// TwinCAT 3 PLC project Katzenhofer
// ProgramVersion: 3.1.4023.0
// libraries:
//   EfficientIO Energy Basic, * (EfficientIO)
//   EfficientIO ModbusTCP, * (EfficientIO)
//   Lynus Persistent Data V1, * (Lynus AG)
//   Lynus Standards, * (EfficientIO)
//   Tc2_IoFunctions, * (Beckhoff Automation GmbH)
//   Tc2_ModbusSrv, * (Beckhoff Automation GmbH)
//   Tc2_Standard, * (Beckhoff Automation GmbH)
//   Tc2_System, * (Beckhoff Automation GmbH)
//   Tc2_Utilities, * (Beckhoff Automation GmbH)
//   Tc3_Module, * (Beckhoff Automation GmbH)
//   EfficientIO Communicator,newest,EfficientIO
// project tree:
//   / FastTask.TcTTO (not stored), MiddleTask.TcTTO, SlowTask.TcTTO
//   FB/ FB_IntervalBit.TcPOU (not stored), FB_ModBus_100Registers_FC3.TcPOU, FB_ModBus_100Registers_FC3_inclID.TcPOU
//   POUs/ prgBattery.TcPOU, prgCalc.TcPOU, prgComEffIO.TcPOU, prgCS.TcPOU, prgEM.TcPOU, prgEMS.TcPOU, prgGrid.TcPOU, prgPersistent.TcPOU, prgPV.TcPOU, prgRWEffIO.TcPOU, prgVarEffIO.TcPOU
// real-time tasks:
//   TASK FastTask: cycle T#5ms, priority 6, ADS port 350
//   TASK MiddleTask: cycle T#10ms, priority 8, ADS port 351
//   TASK SlowTask: cycle T#20ms, priority 10, ADS port 352
// I/O:
//   DEVICE Device 1 (Beckhoff CCAT)
//   DEVICE Device 2 (CX-BK)
//     Box 1 (CX-BK)
// variable links:
//   Katzenhofer/Katzenhofer Instance <-> Device 2 (CX-BK)/Box 1 (CX-BK)
//     MiddleTask Inputs/prgEM.fbEM1.fbKL3403.byStateCH1 <-> Term 2 (KL3403)/Channel 1/State
//     MiddleTask Inputs/prgEM.fbEM1.fbKL3403.byStateCH2 <-> Term 2 (KL3403)/Channel 2/State
//     MiddleTask Inputs/prgEM.fbEM1.fbKL3403.byStateCH3 <-> Term 2 (KL3403)/Channel 3/State
//     MiddleTask Inputs/prgEM.fbEM1.fbKL3403.iDataInCH1 <-> Term 2 (KL3403)/Channel 1/Data In
//     MiddleTask Inputs/prgEM.fbEM1.fbKL3403.iDataInCH2 <-> Term 2 (KL3403)/Channel 2/Data In
//     MiddleTask Inputs/prgEM.fbEM1.fbKL3403.iDataInCH3 <-> Term 2 (KL3403)/Channel 3/Data In
//     MiddleTask Inputs/prgEM.fbKBusState.uiKBusState_OUT <-> Inputs/State
//     MiddleTask Outputs/prgEM.fbEM1.fbKL3403.byCntrCH1 <-> Term 2 (KL3403)/Channel 1/Ctrl
//     MiddleTask Outputs/prgEM.fbEM1.fbKL3403.byCntrCH2 <-> Term 2 (KL3403)/Channel 2/Ctrl
//     MiddleTask Outputs/prgEM.fbEM1.fbKL3403.byCntrCH3 <-> Term 2 (KL3403)/Channel 3/Ctrl

CONFIGURATION Katzenhofer
    RESOURCE PLC ON TwinCAT3
        TASK MiddleTask(INTERVAL := T#10ms, PRIORITY := 8);
        TASK SlowTask(INTERVAL := T#20ms, PRIORITY := 10);
        PROGRAM prgEMS WITH MiddleTask : prgEMS;
        PROGRAM prgPersistent WITH MiddleTask : prgPersistent;
        PROGRAM prgPV WITH MiddleTask : prgPV;
        PROGRAM prgBattery WITH MiddleTask : prgBattery;
        PROGRAM prgEM WITH MiddleTask : prgEM;
        PROGRAM prgGrid WITH MiddleTask : prgGrid;
        PROGRAM prgCS WITH MiddleTask : prgCS;
        PROGRAM prgCalc WITH MiddleTask : prgCalc;
        PROGRAM prgComEffIO WITH SlowTask : prgComEffIO;
    END_RESOURCE
END_CONFIGURATION

// ---- POUs/prgEMS.TcPOU
PROGRAM prgEMS
VAR PERSISTENT
	byMaxDepthOfDischrgEPO		: BYTE;							//{#lynus.ag#()}
	byPrioMinChrgBattSOCInEPO	: BYTE;							//{#lynus.ag#()}
	byResChrgfromGridToBatt		: BYTE;							//{#lynus.ag#()}
	byReserveSOCEPO				: BYTE;							//{#lynus.ag#()}
	uiUpdateTime				: UINT;							//{#lynus.ag#()}
	bEnableEMS					: BOOL;							//{#lynus.ag#()}
	bAllowChrgFromGrid			: BOOL;							//{#lynus.ag#()}
	rMainFuseCSEMS				: REAL;							//{#lynus.ag#()}
	iOperationModeEMS			: INT;							//{#lynus.ag#()}
	by_MinSOC_AdaptiveLC		: BYTE;							//{#lynus.ag#()}
END_VAR
VAR
	fbEMS						: FB_EMS_V12;
	bIsEnableEMS				: BOOL;							//{#lynus.ag#()}
	bStateAllowChrgFromGrid		: BOOL;							//{#lynus.ag#()}
	bHPActivate					: BOOL;							//{#lynus.ag#()}
	bControllingState			: BOOL;							//{#lynus.ag#()}
	iMessageEMS					: INT;							//{#lynus.ag#()}
	rHeartbeatEMS				: REAL;							//{#lynus.ag#()}
	rErrorWarningEMS			: REAL;							//{#lynus.ag#()}
	rReadyEMS					: REAL;							//{#lynus.ag#()}
	rNewBatteryPowerEMS			: REAL;							//{#lynus.ag#()}
	fbRestart					: NT_Reboot;
	byte_test: BYTE;
	real_test: REAL;
	m_test: BOOL;
	lreal_Test: LREAL;
	m_test2: BOOL;
	by_test: BYTE;
	m_Test3: BOOL;
	m_ZeroPowerRegulationActive: BOOL:=FALSE;					//{#lynus.ag#()}
	m_Enable_Dynamic_LM: BOOL;
	timer_CarConnected_CSPowerlow: Ton;
	m_ByteTemp: BOOL;					//{#lynus.ag#()}
	dw_Test: DWORD;
	iOperationModeEMS_actual	: INT;							//{#lynus.ag#()}
END_VAR

fbEMS.stSetupEMS.bAllowChrgFromGrid := bAllowChrgFromGrid;
fbEMS.stSetupEMS.byMaxDepthOfDischrgEPO := byMaxDepthOfDischrgEPO;
fbEMS.stSetupEMS.byPrioMinChrgBattSOCInEPO := byPrioMinChrgBattSOCInEPO;
fbEMS.stSetupEMS.byResChrgfromGridToBatt := byResChrgfromGridToBatt;
fbEMS.stSetupEMS.byReserveSOCEPO := byReserveSOCEPO;
fbEMS.stSetupEMS.rSizeMainFuseCS := rMainFuseCSEMS;
fbEMS.stSetupEMS.uiUpdateTime := uiUpdateTime;


(*
IF m_Enable_Dynamic_LM THEN
	IF prgBattery.dwSOCBattery > byMinSOCdynamicLM AND NOT prgCS.bCarConnected THEN
		iOperationModeEMS := 1;		// Eigenbedarfsoptimierung
	ELSE
		iOperationModeEMS := 3;		// Lastmanagement
	END_IF  
END_IF
*)

IF iOperationModeEMS = 0 THEN fbEMS.eOperationMode_Ext := E_OperatingMode_EMS.eAllOff;
ELSIF iOperationModeEMS = 1 THEN fbEMS.eOperationMode_Ext := E_OperatingMode_EMS.eSelfConsumption;	
ELSIF iOperationModeEMS = 2 THEN fbEMS.eOperationMode_Ext := E_OperatingMode_EMS.ePeakLoadCapping;
ELSIF iOperationModeEMS = 3 THEN fbEMS.eOperationMode_Ext := E_OperatingMode_EMS.eLoadManagement;			
ELSIF iOperationModeEMS = 4 THEN fbEMS.eOperationMode_Ext := E_OperatingMode_EMS.eAdaptiveLoadControl;			

END_IF

fbEMS(
	bEnable:= bEnableEMS, 
	diNrOfEM_IN_ECS:= , 
	stSetupEMS:= , 
	eOperationMode_Ext:= , 
	eSpeedModeBackendController:= E_SpeedModeBackendController_EMS.eSlow, 
	eSpeedModeLocalController:= E_SpeedModeLocalController_EMS.eSlow,
	bZeroPowerRegulation := m_ZeroPowerRegulationActive,
	by_MinSOC_AdaptiveLC:= by_MinSOC_AdaptiveLC , 
	bActivateHP:= bHPActivate, 
	bControllingState:= TRUE, //bControllingState, 
	rHeartbeat:= rHeartbeatEMS, 
	rErrorWarning:= rErrorWarningEMS, 
	rEnergyOptReady:= rReadyEMS, 
	rNewBattPower:= rNewBatteryPowerEMS, 
	b_AnyCarConnected:= prgCS.bCarConnected, 
	eMessageEMS=> iMessageEMS, 
	bStateEnable=> bIsEnableEMS, 
	bStateAllowChrgFromGrid=> bStateAllowChrgFromGrid, 
	bMissingPowerData=> , 
	bSurplusAvailable=> , 
	byProgress=> , 
	uiState_OUT=> , 
	diNrOfEMS_OUT=> , 
	arrMinPrioReached=> , 
	arrMaxPrioReached=> );

	
iOperationModeEMS_actual := fbEMS.eOperationMode;
	
fbRestart(
	NETID:= , 
	DELAY:= , 
	START:= , 
	TMOUT:= , 
	BUSY=> , 
	ERR=> , 
	ERRID=> );
	

timer_CarConnected_CSPowerlow( 	IN := prgCS.bCarConnected AND prgCS.lrPowerCS < 2,	// required to get out of zero power regulation if a car is connected all night long
								PT := T#10M);
							
m_ZeroPowerRegulationActive := prgCS.bCarConnected AND NOT timer_CarConnected_CSPowerlow.Q;
	
// TEMP

real_test:= Lynus_Standards.GVL_Energy.stDataElectricChargingStations[1,1].rTargetPowerEMS;


//byte_test:=Lynus_Standards.GVL_Energy.stDataElectricChargingStations[1,1].byPriority;
 
//m_test:=Lynus_Standards.GVL_Energy.stDataElectricChargingStations[1,1].bEnabled; 
//Lynus_Standards.GVL_Energy.stDataElectricChargingStations[1,1].rTargetPowerEMS 
//Lynus_Standards.GVL_Energy.stDataElectricChargingStations[1,1].rTargetPowerEMS + rValuePercentToControllableDevices;
		
 lreal_Test:=fbEMS.lrPowerDiffFuseECS;
 
m_test2:=Lynus_Standards.GVL_Energy.stDataElectricChargingStations[1,1].bIsControllable;
by_test:=Lynus_Standards.GVL_Energy.stDataElectricChargingStations[1,1].byPriority;
//by_test:=Lynus_Standards.GVL_Energy.stDataElectricChargingStations[1,fbEMS.arrLPPrioZeroSetToZeroP[5]].byPriority;
by_test:= Lynus_Standards.GVL_Energy.stDataElectricChargingStations[1,1].byPriority; 
 
m_Test3:=Lynus_Standards.GVL_Energy.stDataElectricMeters[1].bEnabled ;

END_PROGRAM

// ---- POUs/prgCS.TcPOU
PROGRAM prgCS
VAR PERSISTENT
	bEnabledCS				: BOOL;									//{#lynus.ag#()}
	byPrioCS				: BYTE;									//{#lynus.ag#()}
	bySOC_E_CS				: BYTE;									//{#lynus.ag#()}
	bySOC_D_CS				: BYTE;									//{#lynus.ag#()}
	byMinPowerCS			: BYTE;									//{#lynus.ag#()}
	rMaxPowerCS				: REAL;									//{#lynus.ag#()}
	lrCounterCS				: LREAL;								//{#lynus.ag#()}
	byManualyTargetPower	: BYTE;									//{#lynus.ag#()}
	bManualyOn				: BOOL;									//{#lynus.ag#()}
END_VAR
VAR
	fbCS					: FB_ECS_Alpitronic_Hypercharger;
	fbCSCounter				: FB_EnergyCounter;
	bIsEnabledCS			: BOOL;									//{#lynus.ag#()}
	byErrorWarningCS		: BYTE;									//{#lynus.ag#()}
	byStateMinPowerCS		: BYTE;									//{#lynus.ag#()}
	rTargetPowerCS			: REAL;									//{#lynus.ag#()}
	bCarConnected			: BOOL;									//{#lynus.ag#()}
	rChrgTime				: REAL;									//{#lynus.ag#()}
	lrPowerCS				: LREAL;								//{#lynus.ag#()}
	bSManualyOn				: BOOL;									//{#lynus.ag#()}
	bySManualyTargetPower	: BYTE;									//{#lynus.ag#()}
	b_CS_ModbusFault		: BOOL;									//{#lynus.ag#()}
END_VAR

fbCS.stSetupECS.byDisableSOC := bySOC_D_CS;
fbCS.stSetupECS.byEnableSOC := bySOC_E_CS;
fbCS.stSetupECS.byPriority := byPrioCS;
fbCS.stSetupECS.rMaxPower := rMaxPowerCS;
fbCS.stSetupECS.byCSMinPower := byMinPowerCS;
fbCS.stSetupECS.bManualyOn := bManualyOn;
fbCS.stSetupECS.byManualyTargetPower := byManualyTargetPower;

fbCS(
	bEnable:= bEnabledCS, 
	bPowerDataInvers:= , 
	byUnitID:= 1,				//Allways 1 
	diNrOfEMS_IN:= prgEMS.fbEMS.diNrOfEMS_OUT, 
	diNrOfEM_IN_CS:= , 
	sIPAdress:= '10.11.90.140',			//192.168.0.100', 
	stSetupECS:= , 
	stDataECS=> , 
	diNrOfECS_OUT=> );

bIsEnabledCS := fbCS.stDataECS.bEnabled;
byStateMinPowerCS := fbCS.stDataECS.bySCSMinPower;
rTargetPowerCS := fbCS.stDataECS.rTargetPower;	
byErrorWarningCS := fbCS.stDataECS.byErrorWarning;
bCarConnected := fbCS.stDataECS.bCarConnected;
rChrgTime := fbCS.stDataECS.arrChargingTimeInMin[1];
lrPowerCS := fbCS.stDataECS.lrTotalPower;
bSManualyOn := fbCS.stDataECS.bSManualyOn;
bySManualyTargetPower := fbCS.stDataECS.bySManualyTargetPower;
						
// EnergyCounter
fbCSCounter(
	byActiveTariff:= 1, 
	lrPowerInput:= lrPowerCS, 
	lrTotalCounterEnergy_Consumption=> );
	
IF fbCSCounter.lrTotalCounterEnergy_Consumption > lrCounterCS THEN  	
	lrCounterCS := fbCSCounter.lrTotalCounterEnergy_Consumption;
END_IF

b_CS_ModbusFault := fbCS.bMBTCPError;

END_PROGRAM

// ---- POUs/prgPersistent.TcPOU
PROGRAM prgPersistent
VAR
	fbUSV		: FB_WritePersistentData_CX81xx;

	fb_Reboot		: NT_reboot;
	m_Reboot		: BOOL:=FALSE;

END_VAR

fbUSV(
	eSaveModeData:= eUSVSaveMode.eSaveWhenPowerfail, 
	bLoadPersistentDataOk=> , 
	bPowerFailDetect=> , 
	bError=> , 
	bySaveProcess=> , 
	dwStorageLast24h=> , 
	udiErrorCode=> );
	
	
		
fb_Reboot(	netid := '',
			delay := 2,
			start := m_Reboot);

END_PROGRAM

// ---- POUs/prgPV.TcPOU
PROGRAM prgPV
VAR
	fbPV					: FB_Symo_PV_Inverter_FLOAT_1_DM_30_Inverter;
	fbPV_2					: FB_Symo_PV_Inverter_FLOAT_1_DM_30_Inverter;
	fbPV_3					: FB_Symo_PV_Inverter_FLOAT_1_DM_30_Inverter;
	fbPV_4					: FB_Symo_PV_Inverter_FLOAT_1_DM_30_Inverter;		//Neu
	fbPVInt					: FB_PV_Power;
	fbPVInt_2				: FB_PV_Power;
	fbPVInt_3				: FB_PV_Power;
	fbPVInt_4				: FB_PV_Power;										//Neu
	fbPVCounter				: FB_EnergyCounter;
	fbPVCounter_1			: FB_EnergyCounter;
	fbPVCounter_2			: FB_EnergyCounter;
	fbPVCounter_3			: FB_EnergyCounter;
	fbPVCounter_4			: FB_EnergyCounter;
	fbPVCounter_5			: FB_EnergyCounter;
	fbPVCounter_6			: FB_EnergyCounter;
	fbPVCounter_7			: FB_EnergyCounter;
	fbPVCounter_8			: FB_EnergyCounter;
	fbPVCounter_9			: FB_EnergyCounter;
	fbPVCounter_10			: FB_EnergyCounter;
	fbPVCounter_11			: FB_EnergyCounter;
	fbPVCounter_12			: FB_EnergyCounter;
	fbPVCounter_13			: FB_EnergyCounter;
	fbPVCounter_14			: FB_EnergyCounter;
	fbPVCounter_15			: FB_EnergyCounter;
	fbPVCounter_16			: FB_EnergyCounter;		//Neu
	fbPVCounter_17			: FB_EnergyCounter;		//Neu
	fbPVCounter_18			: FB_EnergyCounter;		//Neu
	fbPVCounter_19			: FB_EnergyCounter;		//Neu
	
	lrPowerPV				: LREAL;				//{#lynus.ag#()}
	byErrorWarningPV		: BYTE;					//{#lynus.ag#()}
	lrPowerPV_1				: LREAL;				//{#lynus.ag#()}
	lrPowerPV_2				: LREAL;				//{#lynus.ag#()}
	lrPowerPV_3				: LREAL;				//{#lynus.ag#()}
	lrPowerPV_4				: LREAL;				//{#lynus.ag#()}
	lrPowerPV_5				: LREAL;				//{#lynus.ag#()}
	lrPowerPV_6				: LREAL;				//{#lynus.ag#()}
	lrPowerPV_7				: LREAL;				//{#lynus.ag#()}
	lrPowerPV_8				: LREAL;				//{#lynus.ag#()}
	lrPowerPV_9				: LREAL;				//{#lynus.ag#()}
	lrPowerPV_10			: LREAL;				//{#lynus.ag#()}
	lrPowerPV_11			: LREAL;				//{#lynus.ag#()}
	lrPowerPV_12			: LREAL;				//{#lynus.ag#()}
	lrPowerPV_13			: LREAL;				//{#lynus.ag#()}
	lrPowerPV_14			: LREAL;				//{#lynus.ag#()}
	lrPowerPV_15			: LREAL;				//{#lynus.ag#()}
	lrPowerPV_16			: LREAL;				//{#lynus.ag#()}
	lrPowerPV_17			: LREAL;				//{#lynus.ag#()}
	lrPowerPV_18			: LREAL;				//{#lynus.ag#()}
	lrPowerPV_19			: LREAL;				//{#lynus.ag#()}
		
	
	
	byte_Fault_PV_1			: BYTE;					//{#lynus.ag#()}
	byte_Fault_PV_2			: BYTE;					//{#lynus.ag#()}
	byte_Fault_PV_3			: BYTE;					//{#lynus.ag#()}
	byte_Fault_PV_4			: BYTE;					//{#lynus.ag#()}
	byte_Fault_PV_5			: BYTE;					//{#lynus.ag#()}
	byte_Fault_PV_6			: BYTE;					//{#lynus.ag#()}
	byte_Fault_PV_7			: BYTE;					//{#lynus.ag#()}
	byte_Fault_PV_8			: BYTE;					//{#lynus.ag#()}
	byte_Fault_PV_9			: BYTE;					//{#lynus.ag#()}
	byte_Fault_PV_10		: BYTE;					//{#lynus.ag#()}
	byte_Fault_PV_11		: BYTE;					//{#lynus.ag#()}
	byte_Fault_PV_12		: BYTE;					//{#lynus.ag#()}
	byte_Fault_PV_13		: BYTE;					//{#lynus.ag#()}
	byte_Fault_PV_14		: BYTE;					//{#lynus.ag#()}
	byte_Fault_PV_15		: BYTE;					//{#lynus.ag#()}
	byte_Fault_PV_16		: BYTE;					//{#lynus.ag#()}
	byte_Fault_PV_17		: BYTE;					//{#lynus.ag#()}
	byte_Fault_PV_18		: BYTE;					//{#lynus.ag#()}
	byte_Fault_PV_19		: BYTE;					//{#lynus.ag#()}
	ton_Delay_Fault			: ARRAY[1..19] OF TON;
	time_PVFaultDelay		: TIME:=T#10S;
	i: INT;
	fb_readOut : FB_ModBus_100Registers_FC3_inclID;	
	usint_ID: USINT;
	Str_Ip: STRING(20);
	w_Adress:WORD;
	usint_Quantity:USINT;
	arrBuffer_FC3				: ARRAY[1..15,1..20] OF WORD;							
	ton_wait_read_out: Ton;
	y: INT;
	z: INT;
	int_Data_Received_old: INT;
	int_readOut:INT;


	m_Enable: BOOL;
	
	udint_Event1_PV1		: UDINT;							//{#lynus.ag#()}
	udint_Event2_PV1		: UDINT;							//{#lynus.ag#()}
	udint_VendorEvent1_PV1	: udint;							//{#lynus.ag#()}
	udint_VendorEvent2_PV1	: udint;							//{#lynus.ag#()}
	udint_VendorEvent3_PV1	: udint;							//{#lynus.ag#()}
	udint_Event1_PV2		: UDINT;							//{#lynus.ag#()}
	udint_Event2_PV2		: UDINT;							//{#lynus.ag#()}
	udint_VendorEvent1_PV2	: udint;							//{#lynus.ag#()}
	udint_VendorEvent2_PV2	: udint;							//{#lynus.ag#()}
	udint_VendorEvent3_PV2	: udint;							//{#lynus.ag#()}
	udint_Event1_PV3		: UDINT;							//{#lynus.ag#()}
	udint_Event2_PV3		: UDINT;							//{#lynus.ag#()}
	udint_VendorEvent1_PV3	: udint;							//{#lynus.ag#()}
	udint_VendorEvent2_PV3	: udint;							//{#lynus.ag#()}
	udint_VendorEvent3_PV3	: udint;							//{#lynus.ag#()}
	udint_Event1_PV4		: UDINT;							//{#lynus.ag#()}
	udint_Event2_PV4		: UDINT;							//{#lynus.ag#()}
	udint_VendorEvent1_PV4	: udint;							//{#lynus.ag#()}
	udint_VendorEvent2_PV4	: udint;							//{#lynus.ag#()}
	udint_VendorEvent3_PV4	: udint;							//{#lynus.ag#()}
	udint_Event1_PV5		: UDINT;							//{#lynus.ag#()}
	udint_Event2_PV5		: UDINT;							//{#lynus.ag#()}
	udint_VendorEvent1_PV5	: udint;							//{#lynus.ag#()}
	udint_VendorEvent2_PV5	: udint;							//{#lynus.ag#()}
	udint_VendorEvent3_PV5	: udint;							//{#lynus.ag#()}
	udint_Event1_PV6		: UDINT;							//{#lynus.ag#()}
	udint_Event2_PV6		: UDINT;							//{#lynus.ag#()}
	udint_VendorEvent1_PV6	: udint;							//{#lynus.ag#()}
	udint_VendorEvent2_PV6	: udint;							//{#lynus.ag#()}
	udint_VendorEvent3_PV6	: udint;							//{#lynus.ag#()}
	udint_Event1_PV7		: UDINT;							//{#lynus.ag#()}
	udint_Event2_PV7		: UDINT;							//{#lynus.ag#()}
	udint_VendorEvent1_PV7	: udint;							//{#lynus.ag#()}
	udint_VendorEvent2_PV7	: udint;							//{#lynus.ag#()}
	udint_VendorEvent3_PV7	: udint;							//{#lynus.ag#()}
	udint_Event1_PV8		: UDINT;							//{#lynus.ag#()}
	udint_Event2_PV8		: UDINT;							//{#lynus.ag#()}
	udint_VendorEvent1_PV8	: udint;							//{#lynus.ag#()}
	udint_VendorEvent2_PV8	: udint;							//{#lynus.ag#()}
	udint_VendorEvent3_PV8	: udint;							//{#lynus.ag#()}
	udint_Event1_PV9		: UDINT;							//{#lynus.ag#()}
	udint_Event2_PV9		: UDINT;							//{#lynus.ag#()}
	udint_VendorEvent1_PV9	: udint;							//{#lynus.ag#()}
	udint_VendorEvent2_PV9	: udint;							//{#lynus.ag#()}
	udint_VendorEvent3_PV9	: udint;							//{#lynus.ag#()}
	udint_Event1_PV10		: udint;							//{#lynus.ag#()}
	udint_Event2_PV10		: udint;							//{#lynus.ag#()}
	udint_VendorEvent1_PV10	: udint;							//{#lynus.ag#()}
	udint_VendorEvent2_PV10	: udint;							//{#lynus.ag#()}
	udint_VendorEvent3_PV10	: udint;							//{#lynus.ag#()}
	udint_Event1_PV11		: udint;							//{#lynus.ag#()}
	udint_Event2_PV11		: udint;							//{#lynus.ag#()}
	udint_VendorEvent1_PV11	: udint;							//{#lynus.ag#()}
	udint_VendorEvent2_PV11	: udint;							//{#lynus.ag#()}
	udint_VendorEvent3_PV11	: udint;							//{#lynus.ag#()}
	udint_Event1_PV12		: udint;							//{#lynus.ag#()}
	udint_Event2_PV12		: udint;							//{#lynus.ag#()}
	udint_VendorEvent1_PV12	: udint;							//{#lynus.ag#()}
	udint_VendorEvent2_PV12	: udint;							//{#lynus.ag#()}
	udint_VendorEvent3_PV12	: udint;							//{#lynus.ag#()}
	udint_Event1_PV13		: udint;							//{#lynus.ag#()}
	udint_Event2_PV13		: udint;							//{#lynus.ag#()}
	udint_VendorEvent1_PV13	: udint;							//{#lynus.ag#()}
	udint_VendorEvent2_PV13	: udint;							//{#lynus.ag#()}
	udint_VendorEvent3_PV13	: udint;							//{#lynus.ag#()}
	udint_Event1_PV14		: udint;							//{#lynus.ag#()}
	udint_Event2_PV14		: udint;							//{#lynus.ag#()}
	udint_VendorEvent1_PV14	: udint;							//{#lynus.ag#()}
	udint_VendorEvent2_PV14	: udint;							//{#lynus.ag#()}
	udint_VendorEvent3_PV14	: udint;							//{#lynus.ag#()}
	udint_Event1_PV15		: udint;							//{#lynus.ag#()}
	udint_Event2_PV15		: udint;							//{#lynus.ag#()}
	udint_VendorEvent1_PV15	: udint;							//{#lynus.ag#()}
	udint_VendorEvent2_PV15	: udint;							//{#lynus.ag#()}
	udint_VendorEvent3_PV15	: UDINT;							//{#lynus.ag#()}
	udint_Event1_PV16		: UDINT;							//{#lynus.ag#()}
	udint_Event2_PV16		: udint;							//{#lynus.ag#()}
	udint_VendorEvent1_PV16	: udint;							//{#lynus.ag#()}
	udint_VendorEvent2_PV16	: udint;							//{#lynus.ag#()}
	udint_VendorEvent3_PV16	: UDINT;							//{#lynus.ag#()}
	udint_Event1_PV17		: UDINT;							//{#lynus.ag#()}
	udint_Event2_PV17		: udint;							//{#lynus.ag#()}
	udint_VendorEvent1_PV17	: udint;							//{#lynus.ag#()}
	udint_VendorEvent2_PV17	: UDINT;							//{#lynus.ag#()}
	udint_VendorEvent3_PV17	: UDINT;							//{#lynus.ag#()}
	udint_Event1_PV18		: UDINT;							//{#lynus.ag#()}
	udint_Event2_PV18		: udint;							//{#lynus.ag#()}
	udint_VendorEvent1_PV18	: udint;							//{#lynus.ag#()}
	udint_VendorEvent2_PV18	: udint;							//{#lynus.ag#()}
	udint_VendorEvent3_PV18	: UDINT;							//{#lynus.ag#()}
	udint_Event1_PV19		: UDINT;							//{#lynus.ag#()}
	udint_Event2_PV19		: udint;							//{#lynus.ag#()}
	udint_VendorEvent1_PV19	: udint;							//{#lynus.ag#()}
	udint_VendorEvent2_PV19	: udint;							//{#lynus.ag#()}
	udint_VendorEvent3_PV19	: UDINT;							//{#lynus.ag#()}
	fbConvertWordToDword		: FB_CV_WORD_TO_DWORD;			//Convert Word to Dword

	w: INT;

	lrPowerPV_temp: LREAL;
	word_1: WORD;
	word_2: WORD;
	udint_Out: DWORD;
	dword_Out3: DWORD;
	

	b_ModbusFault_PV_1		: BOOL;					//{#lynus.ag#()}
	b_ModbusFault_PV_2		: BOOL;					//{#lynus.ag#()}
	b_ModbusFault_PV_3		: BOOL;					//{#lynus.ag#()}
	b_ModbusFault_PV_4		: BOOL;					//{#lynus.ag#()}
	b_ModbusFault_PV_5		: BOOL;					//{#lynus.ag#()}
	b_ModbusFault_PV_6		: BOOL;					//{#lynus.ag#()}
	b_ModbusFault_PV_7		: BOOL;					//{#lynus.ag#()}
	b_ModbusFault_PV_8		: BOOL;					//{#lynus.ag#()}
	b_ModbusFault_PV_9		: BOOL;					//{#lynus.ag#()}
	b_ModbusFault_PV_10		: BOOL;					//{#lynus.ag#()}
	b_ModbusFault_PV_11		: BOOL;					//{#lynus.ag#()}
	b_ModbusFault_PV_12		: BOOL;					//{#lynus.ag#()}
	b_ModbusFault_PV_13		: BOOL;					//{#lynus.ag#()}
	b_ModbusFault_PV_14		: BOOL;					//{#lynus.ag#()}
	b_ModbusFault_PV_15		: BOOL;					//{#lynus.ag#()}
	b_ModbusFault_PV_16		: BOOL;					//{#lynus.ag#()}
	b_ModbusFault_PV_17		: BOOL;					//{#lynus.ag#()}
	b_ModbusFault_PV_18		: BOOL;					//{#lynus.ag#()}
	b_ModbusFault_PV_19		: BOOL;					//{#lynus.ag#()}
	b_ModbusFault_PV_any	: BOOL;					//{#lynus.ag#()}
END_VAR	
VAR PERSISTENT
	lrCounterPV				: LREAL;				//{#lynus.ag#()}
	lrCounterPV_1			: LREAL;				//{#lynus.ag#()}
	lrCounterPV_2			: LREAL;				//{#lynus.ag#()}
	lrCounterPV_3			: LREAL;				//{#lynus.ag#()}
	lrCounterPV_4			: LREAL;				//{#lynus.ag#()}
	lrCounterPV_5			: LREAL;				//{#lynus.ag#()}
	lrCounterPV_6			: LREAL;				//{#lynus.ag#()}
	lrCounterPV_7			: LREAL;				//{#lynus.ag#()}
	lrCounterPV_8			: LREAL;				//{#lynus.ag#()}
	lrCounterPV_9			: LREAL;				//{#lynus.ag#()}
	lrCounterPV_10			: LREAL;				//{#lynus.ag#()}
	lrCounterPV_11			: LREAL;				//{#lynus.ag#()}
	lrCounterPV_12			: LREAL;				//{#lynus.ag#()}
	lrCounterPV_13			: LREAL;				//{#lynus.ag#()}
	lrCounterPV_14			: LREAL;				//{#lynus.ag#()}
	lrCounterPV_15			: LREAL;				//{#lynus.ag#()}
	lrCounterPV_16			: LREAL;				//{#lynus.ag#()}
	lrCounterPV_17			: LREAL;				//{#lynus.ag#()}
	lrCounterPV_18			: LREAL;				//{#lynus.ag#()}
	lrCounterPV_19			: LREAL;				//{#lynus.ag#()}
END_VAR

fbPV.arrUnitID_Inverter[1] := 1;
fbPV.arrUnitID_Inverter[2] := 2;
fbPV.arrUnitID_Inverter[3] := 3;
fbPV.arrUnitID_Inverter[4] := 4;
fbPV.arrUnitID_Inverter[5] := 5;
fbPV.arrUnitID_Inverter[6] := 6;
fbPV.arrUnitID_Inverter[7] := 7;
fbPV.arrUnitID_Inverter[8] := 8;
fbPV.arrUnitID_Inverter[9] := 9;
fbPV.arrUnitID_Inverter[10] := 10;
fbPV.arrUnitID_Inverter[11] := 11;
fbPV.arrUnitID_Inverter[12] := 12;
fbPV.arrUnitID_Inverter[13] := 13;

fbPV(
	bEnable:= TRUE, 
	sIPAdress:= '192.168.0.101', 							//IP-Adresse vom Wechselrichter Master 1 [20.0-3-M](7)
	arrUnitID_Inverter:=  , 
	arrDataSymo10=> , 
	stDataEMPower_PV=> , 
	stDataEMCounter_PV=> , 
	diNrOfEM_OUT_PV=> );

lrPowerPV_1 := fbPV.arrDataSymo10[1].lrPowerAcInverter;
lrPowerPV_2 := fbPV.arrDataSymo10[2].lrPowerAcInverter;
lrPowerPV_3 := fbPV.arrDataSymo10[3].lrPowerAcInverter;
lrPowerPV_4 := fbPV.arrDataSymo10[4].lrPowerAcInverter;
lrPowerPV_5 := fbPV.arrDataSymo10[5].lrPowerAcInverter;
lrPowerPV_6 := fbPV.arrDataSymo10[6].lrPowerAcInverter;
lrPowerPV_7 := fbPV.arrDataSymo10[7].lrPowerAcInverter;
lrPowerPV_8 := fbPV.arrDataSymo10[8].lrPowerAcInverter;
lrPowerPV_9 := fbPV.arrDataSymo10[9].lrPowerAcInverter;
lrPowerPV_10 := fbPV.arrDataSymo10[10].lrPowerAcInverter;
lrPowerPV_11 := fbPV.arrDataSymo10[11].lrPowerAcInverter;
lrPowerPV_12 := fbPV.arrDataSymo10[12].lrPowerAcInverter;
lrPowerPV_13 := fbPV.arrDataSymo10[13].lrPowerAcInverter;

fbPV_2.arrUnitID_Inverter[1] := 1;
fbPV_2(
	bEnable:= TRUE, 
	sIPAdress:= '192.168.0.102', 
	arrUnitID_Inverter:=  , 
	arrDataSymo10=> , 
	stDataEMPower_PV=> , 
	stDataEMCounter_PV=> , 
	diNrOfEM_OUT_PV=> );
lrPowerPV_14 := fbPV_2.arrDataSymo10[1].lrPowerAcInverter;

fbPV_3.arrUnitID_Inverter[1] := 1;
fbPV_3(
	bEnable:= TRUE, 
	sIPAdress:= '192.168.0.103', 
	arrUnitID_Inverter:=  , 
	arrDataSymo10=> , 
	stDataEMPower_PV=> , 
	stDataEMCounter_PV=> , 
	diNrOfEM_OUT_PV=> );
lrPowerPV_15 := fbPV_3.arrDataSymo10[1].lrPowerAcInverter;

// Wohngebaeude 2024
fbPV_4.arrUnitID_Inverter[1] := 1;
fbPV_4.arrUnitID_Inverter[2] := 2;
fbPV_4.arrUnitID_Inverter[3] := 3;
fbPV_4.arrUnitID_Inverter[4] := 4;
fbPV_4(
	bEnable:= TRUE, 
	sIPAdress:= '192.168.0.104', 								//IP-Adresse von Wechselrichter Master 2
	arrUnitID_Inverter:=  , 
	arrDataSymo10=> , 
	stDataEMPower_PV=> , 
	stDataEMCounter_PV=> , 
	diNrOfEM_OUT_PV=> );
	
lrPowerPV_16 := fbPV_4.arrDataSymo10[1].lrPowerAcInverter;
lrPowerPV_17 := fbPV_4.arrDataSymo10[2].lrPowerAcInverter;
lrPowerPV_18 := fbPV_4.arrDataSymo10[3].lrPowerAcInverter;
lrPowerPV_19 := fbPV_4.arrDataSymo10[4].lrPowerAcInverter;

fbPVInt(
	bEnable:= TRUE, 
	bPowerDataInvers:= , 
	diNrOfEM_IN_PV:= fbPV.diNrOfEM_OUT_PV, 
	stDataPv=> , 
	diNrOfPv_OUT=> );
fbPVInt_2(
	bEnable:= TRUE, 
	bPowerDataInvers:= , 
	diNrOfEM_IN_PV:= fbPV_2.diNrOfEM_OUT_PV, 
	stDataPv=> , 
	diNrOfPv_OUT=> );
fbPVInt_3(
	bEnable:= TRUE, 
	bPowerDataInvers:= , 
	diNrOfEM_IN_PV:= fbPV_3.diNrOfEM_OUT_PV, 
	stDataPv=> , 
	diNrOfPv_OUT=> );
fbPVInt_4(
	bEnable:= TRUE, 
	bPowerDataInvers:= , 
	diNrOfEM_IN_PV:= fbPV_4.diNrOfEM_OUT_PV, 
	stDataPv=> , 
	diNrOfPv_OUT=> );


lrPowerPV_temp := fbPVInt.stDataPv.lrPower +  fbPVInt_2.stDataPv.lrPower +  fbPVInt_3.stDataPv.lrPower;
byErrorWarningPV := fbPVInt.stDataPv.byErrorWarning OR fbPVInt_2.stDataPv.byErrorWarning OR fbPVInt_3.stDataPv.byErrorWarning;

lrPowerPV := lrPowerPV_1 + lrPowerPV_2 + lrPowerPV_3 + lrPowerPV_4 + lrPowerPV_5 + lrPowerPV_6 + lrPowerPV_7 + lrPowerPV_8 + lrPowerPV_9 + lrPowerPV_10 + lrPowerPV_11 + lrPowerPV_12 + lrPowerPV_13; // 14+15 auf eigener Einspeisung   + lrPowerPV_14 + lrPowerPV_15 + lrPowerPV_16 + lrPowerPV_17 + lrPowerPV_18 + lrPowerPV_19; 16 bis 19 von den neuen Wechselrichtern


// EnergyCounter Total
fbPVCounter(
	byActiveTariff:= 1, 
	lrPowerInput:= 0 - lrPowerPV, 
	lrTotalCounterEnergy_Consumption=> , 
	lrTotalCounterEnergy_Production=> , 
	lrCounterEnergyT1_Consumption=> , 
	lrCounterEnergyT2_Consumption=> , 
	lrCounterEnergyT1_Production=> , 
	lrCounterEnergyT2_Production=> );
	
IF fbPVCounter.lrTotalCounterEnergy_Production > lrCounterPV THEN  	
	lrCounterPV := fbPVCounter.lrTotalCounterEnergy_Production;
END_IF

// EnergyCounter Separated
fbPVCounter_1(
	byActiveTariff:= 1, 
	lrPowerInput:= 0 - lrPowerPV_1, 
	lrTotalCounterEnergy_Production=> );
	
fbPVCounter_2(
	byActiveTariff:= 1, 
	lrPowerInput:= 0 - lrPowerPV_2, 
	lrTotalCounterEnergy_Production=> );
	
fbPVCounter_3(
	byActiveTariff:= 1, 
	lrPowerInput:= 0 - lrPowerPV_3, 
	lrTotalCounterEnergy_Production=> );
	
fbPVCounter_4(
	byActiveTariff:= 1, 
	lrPowerInput:= 0 - lrPowerPV_4, 
	lrTotalCounterEnergy_Production=> );
	
fbPVCounter_5(
	byActiveTariff:= 1, 
	lrPowerInput:= 0 - lrPowerPV_5, 
	lrTotalCounterEnergy_Production=> );
	
fbPVCounter_6(
	byActiveTariff:= 1, 
	lrPowerInput:= 0 - lrPowerPV_6, 
	lrTotalCounterEnergy_Production=> );
	
fbPVCounter_7(
	byActiveTariff:= 1, 
	lrPowerInput:= 0 - lrPowerPV_7, 
	lrTotalCounterEnergy_Production=> );
	
fbPVCounter_8(
	byActiveTariff:= 1, 
	lrPowerInput:= 0 - lrPowerPV_8, 
	lrTotalCounterEnergy_Production=> );
	
fbPVCounter_9(
	byActiveTariff:= 1, 
	lrPowerInput:= 0 - lrPowerPV_9, 
	lrTotalCounterEnergy_Production=> );
	
fbPVCounter_10(
	byActiveTariff:= 1, 
	lrPowerInput:= 0 - lrPowerPV_10, 
	lrTotalCounterEnergy_Production=> );
	
fbPVCounter_11(
	byActiveTariff:= 1, 
	lrPowerInput:= 0 - lrPowerPV_11, 
	lrTotalCounterEnergy_Production=> );

fbPVCounter_12(
	byActiveTariff:= 1, 
	lrPowerInput:= 0 - lrPowerPV_12, 
	lrTotalCounterEnergy_Production=> );

fbPVCounter_13(
	byActiveTariff:= 1, 
	lrPowerInput:= 0 - lrPowerPV_13, 
	lrTotalCounterEnergy_Production=> );

fbPVCounter_14(
	byActiveTariff:= 1, 
	lrPowerInput:= 0 - lrPowerPV_14, 
	lrTotalCounterEnergy_Production=> );	

fbPVCounter_15(
	byActiveTariff:= 1, 
	lrPowerInput:= 0 - lrPowerPV_15, 
	lrTotalCounterEnergy_Production=> );
	
fbPVCounter_16(
	byActiveTariff:= 1, 
	lrPowerInput:= 0 - lrPowerPV_16, 
	lrTotalCounterEnergy_Production=> );
	
fbPVCounter_17(
	byActiveTariff:= 1, 
	lrPowerInput:= 0 - lrPowerPV_17, 
	lrTotalCounterEnergy_Production=> );
	
fbPVCounter_18(
	byActiveTariff:= 1, 
	lrPowerInput:= 0 - lrPowerPV_18, 
	lrTotalCounterEnergy_Production=> );
	
fbPVCounter_19(
	byActiveTariff:= 1, 
	lrPowerInput:= 0 - lrPowerPV_19, 
	lrTotalCounterEnergy_Production=> );
	
	

	
IF fbPVCounter_1.lrTotalCounterEnergy_Production > lrCounterPV_1 THEN  	
	lrCounterPV_1 := fbPVCounter_1.lrTotalCounterEnergy_Production;
END_IF
IF fbPVCounter_2.lrTotalCounterEnergy_Production > lrCounterPV_2 THEN  	
	lrCounterPV_2 := fbPVCounter_2.lrTotalCounterEnergy_Production;
END_IF
IF fbPVCounter_3.lrTotalCounterEnergy_Production > lrCounterPV_3 THEN  	
	lrCounterPV_3 := fbPVCounter_3.lrTotalCounterEnergy_Production;
END_IF
IF fbPVCounter_4.lrTotalCounterEnergy_Production > lrCounterPV_4 THEN  	
	lrCounterPV_4 := fbPVCounter_4.lrTotalCounterEnergy_Production;
END_IF
IF fbPVCounter_5.lrTotalCounterEnergy_Production > lrCounterPV_5 THEN  	
	lrCounterPV_5 := fbPVCounter_5.lrTotalCounterEnergy_Production;
END_IF
IF fbPVCounter_6.lrTotalCounterEnergy_Production > lrCounterPV_6 THEN  	
	lrCounterPV_6 := fbPVCounter_6.lrTotalCounterEnergy_Production;
END_IF
IF fbPVCounter_7.lrTotalCounterEnergy_Production > lrCounterPV_7 THEN  	
	lrCounterPV_7 := fbPVCounter_7.lrTotalCounterEnergy_Production;
END_IF
IF fbPVCounter_8.lrTotalCounterEnergy_Production > lrCounterPV_8 THEN  	
	lrCounterPV_8 := fbPVCounter_8.lrTotalCounterEnergy_Production;
END_IF
IF fbPVCounter_9.lrTotalCounterEnergy_Production > lrCounterPV_9 THEN  	
	lrCounterPV_9 := fbPVCounter_9.lrTotalCounterEnergy_Production;
END_IF
IF fbPVCounter_10.lrTotalCounterEnergy_Production > lrCounterPV_10 THEN  	
	lrCounterPV_10 := fbPVCounter_10.lrTotalCounterEnergy_Production;
END_IF
IF fbPVCounter_11.lrTotalCounterEnergy_Production > lrCounterPV_11 THEN  	
	lrCounterPV_11 := fbPVCounter_11.lrTotalCounterEnergy_Production;
END_IF
IF fbPVCounter_12.lrTotalCounterEnergy_Production > lrCounterPV_12 THEN  	
	lrCounterPV_12 := fbPVCounter_11.lrTotalCounterEnergy_Production;
END_IF
IF fbPVCounter_13.lrTotalCounterEnergy_Production > lrCounterPV_13 THEN  	
	lrCounterPV_13 := fbPVCounter_11.lrTotalCounterEnergy_Production;
END_IF
IF fbPVCounter_14.lrTotalCounterEnergy_Production > lrCounterPV_14 THEN  	
	lrCounterPV_14 := fbPVCounter_11.lrTotalCounterEnergy_Production;
END_IF
IF fbPVCounter_15.lrTotalCounterEnergy_Production > lrCounterPV_15 THEN  	
	lrCounterPV_15 := fbPVCounter_11.lrTotalCounterEnergy_Production;
END_IF
IF fbPVCounter_16.lrTotalCounterEnergy_Production > lrCounterPV_16 THEN  	
	lrCounterPV_16 := fbPVCounter_11.lrTotalCounterEnergy_Production;
END_IF
IF fbPVCounter_17.lrTotalCounterEnergy_Production > lrCounterPV_17 THEN  	
	lrCounterPV_17 := fbPVCounter_11.lrTotalCounterEnergy_Production;
END_IF
IF fbPVCounter_18.lrTotalCounterEnergy_Production > lrCounterPV_18 THEN  	
	lrCounterPV_18 := fbPVCounter_11.lrTotalCounterEnergy_Production;
END_IF
IF fbPVCounter_19.lrTotalCounterEnergy_Production > lrCounterPV_19 THEN  	
	lrCounterPV_19 := fbPVCounter_11.lrTotalCounterEnergy_Production;
END_IF


// PV inverter Fault Bits
// arrDataSymo10[byInverterInProgress].eOperatingStateInverter := E_Symo_PV_OperatingState.eFaults;


FOR i:= 1 TO 15 BY 1 DO
	ton_Delay_Fault[i](pt := time_PVFaultDelay);
END_FOR
ton_Delay_Fault[1].IN	:=	fbPV.arrDataSymo10[1].eOperatingStateInverter = E_Symo_PV_OperatingState.eFaults OR fbPV.arrDataSymo10[1].eOperatingStateInverter = E_Symo_PV_OperatingState.eNoDataReceived;
ton_Delay_Fault[2].IN	:=	fbPV.arrDataSymo10[2].eOperatingStateInverter = E_Symo_PV_OperatingState.eFaults OR fbPV.arrDataSymo10[2].eOperatingStateInverter = E_Symo_PV_OperatingState.eNoDataReceived;
ton_Delay_Fault[3].IN	:=	fbPV.arrDataSymo10[3].eOperatingStateInverter = E_Symo_PV_OperatingState.eFaults OR fbPV.arrDataSymo10[3].eOperatingStateInverter = E_Symo_PV_OperatingState.eNoDataReceived;
ton_Delay_Fault[4].IN	:=	fbPV.arrDataSymo10[4].eOperatingStateInverter = E_Symo_PV_OperatingState.eFaults OR fbPV.arrDataSymo10[4].eOperatingStateInverter = E_Symo_PV_OperatingState.eNoDataReceived;
ton_Delay_Fault[5].IN	:=	fbPV.arrDataSymo10[5].eOperatingStateInverter = E_Symo_PV_OperatingState.eFaults OR fbPV.arrDataSymo10[5].eOperatingStateInverter = E_Symo_PV_OperatingState.eNoDataReceived;
ton_Delay_Fault[6].IN	:=	fbPV.arrDataSymo10[6].eOperatingStateInverter = E_Symo_PV_OperatingState.eFaults OR fbPV.arrDataSymo10[6].eOperatingStateInverter = E_Symo_PV_OperatingState.eNoDataReceived;
ton_Delay_Fault[7].IN	:=	fbPV.arrDataSymo10[7].eOperatingStateInverter = E_Symo_PV_OperatingState.eFaults OR fbPV.arrDataSymo10[7].eOperatingStateInverter = E_Symo_PV_OperatingState.eNoDataReceived;
ton_Delay_Fault[8].IN	:=	fbPV.arrDataSymo10[8].eOperatingStateInverter = E_Symo_PV_OperatingState.eFaults OR fbPV.arrDataSymo10[8].eOperatingStateInverter = E_Symo_PV_OperatingState.eNoDataReceived;
ton_Delay_Fault[9].IN	:=	fbPV.arrDataSymo10[9].eOperatingStateInverter = E_Symo_PV_OperatingState.eFaults OR fbPV.arrDataSymo10[9].eOperatingStateInverter = E_Symo_PV_OperatingState.eNoDataReceived;
ton_Delay_Fault[10].IN	:=	fbPV.arrDataSymo10[10].eOperatingStateInverter = E_Symo_PV_OperatingState.eFaults OR fbPV.arrDataSymo10[10].eOperatingStateInverter = E_Symo_PV_OperatingState.eNoDataReceived;
ton_Delay_Fault[11].IN	:=	fbPV.arrDataSymo10[11].eOperatingStateInverter = E_Symo_PV_OperatingState.eFaults OR fbPV.arrDataSymo10[11].eOperatingStateInverter = E_Symo_PV_OperatingState.eNoDataReceived;
ton_Delay_Fault[12].IN	:=	fbPV.arrDataSymo10[12].eOperatingStateInverter = E_Symo_PV_OperatingState.eFaults OR fbPV.arrDataSymo10[12].eOperatingStateInverter = E_Symo_PV_OperatingState.eNoDataReceived;
ton_Delay_Fault[13].IN	:=	fbPV.arrDataSymo10[13].eOperatingStateInverter = E_Symo_PV_OperatingState.eFaults OR fbPV.arrDataSymo10[13].eOperatingStateInverter = E_Symo_PV_OperatingState.eNoDataReceived;
ton_Delay_Fault[14].IN	:=	fbPV_2.arrDataSymo10[1].eOperatingStateInverter = E_Symo_PV_OperatingState.eFaults OR fbPV_2.arrDataSymo10[1].eOperatingStateInverter = E_Symo_PV_OperatingState.eNoDataReceived;
ton_Delay_Fault[15].IN	:=	fbPV_3.arrDataSymo10[1].eOperatingStateInverter = E_Symo_PV_OperatingState.eFaults OR fbPV_3.arrDataSymo10[1].eOperatingStateInverter = E_Symo_PV_OperatingState.eNoDataReceived;
ton_Delay_Fault[16].IN	:=	fbPV_4.arrDataSymo10[1].eOperatingStateInverter = E_Symo_PV_OperatingState.eFaults OR fbPV_4.arrDataSymo10[1].eOperatingStateInverter = E_Symo_PV_OperatingState.eNoDataReceived;
ton_Delay_Fault[17].IN	:=	fbPV_4.arrDataSymo10[2].eOperatingStateInverter = E_Symo_PV_OperatingState.eFaults OR fbPV_4.arrDataSymo10[2].eOperatingStateInverter = E_Symo_PV_OperatingState.eNoDataReceived;
ton_Delay_Fault[18].IN	:=	fbPV_4.arrDataSymo10[3].eOperatingStateInverter = E_Symo_PV_OperatingState.eFaults OR fbPV_4.arrDataSymo10[3].eOperatingStateInverter = E_Symo_PV_OperatingState.eNoDataReceived;
ton_Delay_Fault[19].IN	:=	fbPV_4.arrDataSymo10[4].eOperatingStateInverter = E_Symo_PV_OperatingState.eFaults OR fbPV_4.arrDataSymo10[4].eOperatingStateInverter = E_Symo_PV_OperatingState.eNoDataReceived;


(*
Byte_Fault_PV_1		:=	2 * BOOL_TO_BYTE(ton_Delay_Fault[1].Q);
Byte_Fault_PV_2		:=	2 * BOOL_TO_BYTE(ton_Delay_Fault[2].Q);
Byte_Fault_PV_3		:=	2 * BOOL_TO_BYTE(ton_Delay_Fault[3].Q);
Byte_Fault_PV_4		:=	2 * BOOL_TO_BYTE(ton_Delay_Fault[4].Q);
Byte_Fault_PV_5		:=	2 * BOOL_TO_BYTE(ton_Delay_Fault[5].Q);
Byte_Fault_PV_6		:=	2 * BOOL_TO_BYTE(ton_Delay_Fault[6].Q);
Byte_Fault_PV_7		:=	2 * BOOL_TO_BYTE(ton_Delay_Fault[7].Q);
Byte_Fault_PV_8		:=	2 * BOOL_TO_BYTE(ton_Delay_Fault[8].Q);
Byte_Fault_PV_9		:=	2 * BOOL_TO_BYTE(ton_Delay_Fault[9].Q);
Byte_Fault_PV_10	:=	2 * BOOL_TO_BYTE(ton_Delay_Fault[10].Q);
Byte_Fault_PV_11	:=  2 * BOOL_TO_BYTE(ton_Delay_Fault[11].Q);
Byte_Fault_PV_12	:=	2 * BOOL_TO_BYTE(ton_Delay_Fault[12].Q);
Byte_Fault_PV_13	:=	2 * BOOL_TO_BYTE(ton_Delay_Fault[13].Q);
Byte_Fault_PV_14	:=	2 * BOOL_TO_BYTE(ton_Delay_Fault[14].Q);
Byte_Fault_PV_15	:=	2 * BOOL_TO_BYTE(ton_Delay_Fault[15].Q);

*)


// read out event registers
IF NOT m_Enable THEN 
	int_readOut := -1;
END_IF
CASE int_readOut OF
	0: // wait state
		fb_readOut.m_Enable := FALSE;
		ton_wait_read_out.IN := TRUE;
		IF ton_wait_read_out.Q THEN
			ton_wait_read_out.IN := FALSE;
			int_readOut := int_readOut +1;
		END_IF
	1: // read out IP 192.168.0.101 ID1  PV1 
		fb_readOut.m_Enable := TRUE;
		Str_Ip := '192.168.0.101';
		usint_Quantity := 16;
		w_Adress := 40117;
		usint_ID := 1;
		int_readOut := int_readOut +1;
	2: // wait for received values	
		ton_wait_read_out.IN := TRUE;
		IF NOT fb_readOut.fbMBRead_FC3.bBusy AND int_Data_Received_old <> fb_readout.int_Data_Received  THEN
			y:=1;
			FOR z:=1 TO 20 BY 1 DO
				arrBuffer_FC3[y,z] := fb_readOut.w_Array_Received[z];
			END_FOR
			fb_readOut.m_Enable := FALSE;
			ton_wait_read_out.IN := FALSE;
			int_readOut := int_readOut +1;	
		ELSIF fb_readOut.fbMBRead_FC3.bError THEN
			fb_readOut.m_Enable := FALSE;
			ton_wait_read_out.IN := FALSE;
			int_readOut := int_readOut +1;		
		ELSIF ton_wait_read_out.Q THEN
			fb_readOut.m_Enable := FALSE;
			ton_wait_read_out.IN := FALSE;
			int_readOut := int_readOut +1;		
		END_IF
	3: // wait state
		fb_readOut.m_Enable := FALSE;
		ton_wait_read_out.IN := TRUE;
		IF ton_wait_read_out.Q THEN
			ton_wait_read_out.IN := FALSE;
			int_readOut := int_readOut +1;
		END_IF
	4: // read out IP 192.168.0.101 ID2   PV2 
		fb_readOut.m_Enable := TRUE;
		Str_Ip := '192.168.0.101';
		usint_ID := 2;
		int_Data_Received_old := fb_readout.int_Data_Received;
		int_readOut := int_readOut +1;
	5: // wait for received values	
		ton_wait_read_out.IN := TRUE;
		IF NOT fb_readOut.fbMBRead_FC3.bBusy AND int_Data_Received_old <> fb_readout.int_Data_Received  THEN
			y:=2;
			FOR z:=1 TO 20 BY 1 DO
				arrBuffer_FC3[y,z] := fb_readOut.w_Array_Received[z];
			END_FOR
			fb_readOut.m_Enable := FALSE;
			ton_wait_read_out.IN := FALSE;
			int_readOut := int_readOut +1;	
		ELSIF fb_readOut.fbMBRead_FC3.bError THEN
			fb_readOut.m_Enable := FALSE;
			ton_wait_read_out.IN := FALSE;
			int_readOut := int_readOut +1;		
		ELSIF ton_wait_read_out.Q THEN
			fb_readOut.m_Enable := FALSE;
			ton_wait_read_out.IN := FALSE;
			int_readOut := int_readOut +1;		
		END_IF
	6: // wait state
		fb_readOut.m_Enable := FALSE;
		ton_wait_read_out.IN := TRUE;
		IF ton_wait_read_out.Q THEN
			ton_wait_read_out.IN := FALSE;
			int_readOut := int_readOut +1;
		END_IF
	7: // read out IP 192.168.0.101  ID3 PV3 
		fb_readOut.m_Enable := TRUE;
		Str_Ip := '192.168.0.101';
		usint_ID := 3;
		int_readOut := int_readOut +1;
	8: // wait for received values	
		ton_wait_read_out.IN := TRUE;
		IF NOT fb_readOut.fbMBRead_FC3.bBusy AND int_Data_Received_old <> fb_readout.int_Data_Received  THEN
			y:=3;
			FOR z:=1 TO 20 BY 1 DO
				arrBuffer_FC3[y,z] := fb_readOut.w_Array_Received[z];
			END_FOR
			fb_readOut.m_Enable := FALSE;
			ton_wait_read_out.IN := FALSE;
			int_readOut := int_readOut +1;	
		ELSIF fb_readOut.fbMBRead_FC3.bError THEN
			fb_readOut.m_Enable := FALSE;
			ton_wait_read_out.IN := FALSE;
			int_readOut := int_readOut +1;		
		ELSIF ton_wait_read_out.Q THEN
			fb_readOut.m_Enable := FALSE;
			ton_wait_read_out.IN := FALSE;
			int_readOut := int_readOut +1;		
		END_IF
	9: // wait state
		fb_readOut.m_Enable := FALSE;
		ton_wait_read_out.IN := TRUE;
		IF ton_wait_read_out.Q THEN
			ton_wait_read_out.IN := FALSE;
			int_readOut := int_readOut +1;
		END_IF
	10: // read out IP 192.168.0.101 ID4  PV4 
		fb_readOut.m_Enable := TRUE;
		Str_Ip := '192.168.0.101';
		usint_ID := 4;
		int_Data_Received_old := fb_readout.int_Data_Received;
		int_readOut := int_readOut +1;
	11: // wait for received values	
		ton_wait_read_out.IN := TRUE;
		IF NOT fb_readOut.fbMBRead_FC3.bBusy AND int_Data_Received_old <> fb_readout.int_Data_Received  THEN
			y:=4;
			FOR z:=1 TO 20 BY 1 DO
				arrBuffer_FC3[y,z] := fb_readOut.w_Array_Received[z];
			END_FOR
			fb_readOut.m_Enable := FALSE;
			ton_wait_read_out.IN := FALSE;
			int_readOut := int_readOut +1;	
		ELSIF fb_readOut.fbMBRead_FC3.bError THEN
			fb_readOut.m_Enable := FALSE;
			ton_wait_read_out.IN := FALSE;
			int_readOut := int_readOut +1;		
		ELSIF ton_wait_read_out.Q THEN
			fb_readOut.m_Enable := FALSE;
			ton_wait_read_out.IN := FALSE;
			int_readOut := int_readOut +1;		
		END_IF
	12: // wait state
		fb_readOut.m_Enable := FALSE;
		ton_wait_read_out.IN := TRUE;
		IF ton_wait_read_out.Q THEN
			ton_wait_read_out.IN := FALSE;
			int_readOut := int_readOut +1;
		END_IF
	13: // read out IP 192.168.0.101 ID 5  PV5
		fb_readOut.m_Enable := TRUE;
		Str_Ip := '192.168.0.101';
		usint_ID := 5;
		int_Data_Received_old := fb_readout.int_Data_Received;
		int_readOut := int_readOut +1;
	14: // wait for received values	
		ton_wait_read_out.IN := TRUE;
		IF NOT fb_readOut.fbMBRead_FC3.bBusy AND int_Data_Received_old <> fb_readout.int_Data_Received  THEN
			y:=5;
			FOR z:=1 TO 20 BY 1 DO
				arrBuffer_FC3[y,z] := fb_readOut.w_Array_Received[z];
			END_FOR
			fb_readOut.m_Enable := FALSE;
			ton_wait_read_out.IN := FALSE;
			int_readOut := int_readOut +1;	
		ELSIF fb_readOut.fbMBRead_FC3.bError THEN
			fb_readOut.m_Enable := FALSE;
			ton_wait_read_out.IN := FALSE;
			int_readOut := int_readOut +1;		
		ELSIF ton_wait_read_out.Q THEN
			fb_readOut.m_Enable := FALSE;
			ton_wait_read_out.IN := FALSE;
			int_readOut := int_readOut +1;		
		END_IF
	15: // wait state
		fb_readOut.m_Enable := FALSE;
		ton_wait_read_out.IN := TRUE;
		IF ton_wait_read_out.Q THEN
			ton_wait_read_out.IN := FALSE;
			int_readOut := int_readOut +1;
		END_IF	
	16: // read out IP 192.168.0.101 ID 6 PV6  
		fb_readOut.m_Enable := TRUE;
		Str_Ip := '192.168.0.101';
		usint_ID := 6;
		int_Data_Received_old := fb_readout.int_Data_Received;
		int_readOut := int_readOut +1;
	17: // wait for received values	
		ton_wait_read_out.IN := TRUE;
		IF NOT fb_readOut.fbMBRead_FC3.bBusy AND int_Data_Received_old <> fb_readout.int_Data_Received  THEN
			y:=6;
			FOR z:=1 TO 20 BY 1 DO
				arrBuffer_FC3[y,z] := fb_readOut.w_Array_Received[z];
			END_FOR
			fb_readOut.m_Enable := FALSE;
			ton_wait_read_out.IN := FALSE;
			int_readOut := int_readOut +1;	
		ELSIF fb_readOut.fbMBRead_FC3.bError THEN
			fb_readOut.m_Enable := FALSE;
			ton_wait_read_out.IN := FALSE;
			int_readOut := int_readOut +1;		
		ELSIF ton_wait_read_out.Q THEN
			fb_readOut.m_Enable := FALSE;
			ton_wait_read_out.IN := FALSE;
			int_readOut := int_readOut +1;		
		END_IF	
	18: // wait state
		fb_readOut.m_Enable := FALSE;
		ton_wait_read_out.IN := TRUE;
		IF ton_wait_read_out.Q THEN
			ton_wait_read_out.IN := FALSE;
			int_readOut := int_readOut +1;
		END_IF		
	19: // read out IP 192.168.0.101 ID7  PV7 
		fb_readOut.m_Enable := TRUE;
		Str_Ip := '192.168.0.101';
		usint_ID := 7;
		int_Data_Received_old := fb_readout.int_Data_Received;
		int_readOut := int_readOut +1;
	20: // wait for received values	
		ton_wait_read_out.IN := TRUE;
		IF NOT fb_readOut.fbMBRead_FC3.bBusy AND int_Data_Received_old <> fb_readout.int_Data_Received  THEN
			y:=7;
			FOR z:=1 TO 20 BY 1 DO
				arrBuffer_FC3[y,z] := fb_readOut.w_Array_Received[z];
			END_FOR
			fb_readOut.m_Enable := FALSE;
			ton_wait_read_out.IN := FALSE;
			int_readOut := int_readOut +1;	
		ELSIF fb_readOut.fbMBRead_FC3.bError THEN
			fb_readOut.m_Enable := FALSE;
			ton_wait_read_out.IN := FALSE;
			int_readOut := int_readOut +1;		
		ELSIF ton_wait_read_out.Q THEN
			fb_readOut.m_Enable := FALSE;
			ton_wait_read_out.IN := FALSE;
			int_readOut := int_readOut +1;		
		END_IF			
	21: // wait state
		fb_readOut.m_Enable := FALSE;
		ton_wait_read_out.IN := TRUE;
		IF ton_wait_read_out.Q THEN
			ton_wait_read_out.IN := FALSE;
			int_readOut := int_readOut +1;
		END_IF			
	22: // read out IP 192.168.0.101 ID8  PV8 
		fb_readOut.m_Enable := TRUE;
		Str_Ip := '192.168.0.101';
		usint_ID := 8;
		int_Data_Received_old := fb_readout.int_Data_Received;
		int_readOut := int_readOut +1;
	23: // wait for received values	
		ton_wait_read_out.IN := TRUE;
		IF NOT fb_readOut.fbMBRead_FC3.bBusy AND int_Data_Received_old <> fb_readout.int_Data_Received  THEN
			y:=8;
			FOR z:=1 TO 20 BY 1 DO
				arrBuffer_FC3[y,z] := fb_readOut.w_Array_Received[z];
			END_FOR
			fb_readOut.m_Enable := FALSE;
			ton_wait_read_out.IN := FALSE;
			int_readOut := int_readOut +1;	
		ELSIF fb_readOut.fbMBRead_FC3.bError THEN
			fb_readOut.m_Enable := FALSE;
			ton_wait_read_out.IN := FALSE;
			int_readOut := int_readOut +1;		
		ELSIF ton_wait_read_out.Q THEN
			fb_readOut.m_Enable := FALSE;
			ton_wait_read_out.IN := FALSE;
			int_readOut := int_readOut +1;		
		END_IF			
	24: // wait state
		fb_readOut.m_Enable := FALSE;
		ton_wait_read_out.IN := TRUE;
		IF ton_wait_read_out.Q THEN
			ton_wait_read_out.IN := FALSE;
			int_readOut := int_readOut +1;
		END_IF			
	25: // read out IP 192.168.0.101 ID9  PV9 
		fb_readOut.m_Enable := TRUE;
		Str_Ip := '192.168.0.101';
		usint_ID := 9;
		int_Data_Received_old := fb_readout.int_Data_Received;
		int_readOut := int_readOut +1;
	26: // wait for received values	
		ton_wait_read_out.IN := TRUE;
		IF NOT fb_readOut.fbMBRead_FC3.bBusy AND int_Data_Received_old <> fb_readout.int_Data_Received  THEN
			y:=9;
			FOR z:=1 TO 20 BY 1 DO
				arrBuffer_FC3[y,z] := fb_readOut.w_Array_Received[z];
			END_FOR
			fb_readOut.m_Enable := FALSE;
			ton_wait_read_out.IN := FALSE;
			int_readOut := int_readOut +1;	
		ELSIF fb_readOut.fbMBRead_FC3.bError THEN
			fb_readOut.m_Enable := FALSE;
			ton_wait_read_out.IN := FALSE;
			int_readOut := int_readOut +1;		
		ELSIF ton_wait_read_out.Q THEN
			fb_readOut.m_Enable := FALSE;
			ton_wait_read_out.IN := FALSE;
			int_readOut := int_readOut +1;		
		END_IF			
	27: // wait state
		fb_readOut.m_Enable := FALSE;
		ton_wait_read_out.IN := TRUE;
		IF ton_wait_read_out.Q THEN
			ton_wait_read_out.IN := FALSE;
			int_readOut := int_readOut +1;
		END_IF			
	28: // read out IP 192.168.0.101 ID10  PV10 
		fb_readOut.m_Enable := TRUE;
		Str_Ip := '192.168.0.101';
		usint_ID := 10;
		int_Data_Received_old := fb_readout.int_Data_Received;
		int_readOut := int_readOut +1;
	29: // wait for received values	
		ton_wait_read_out.IN := TRUE;
		IF NOT fb_readOut.fbMBRead_FC3.bBusy AND int_Data_Received_old <> fb_readout.int_Data_Received  THEN
			y:=10;
			FOR z:=1 TO 20 BY 1 DO
				arrBuffer_FC3[y,z] := fb_readOut.w_Array_Received[z];
			END_FOR
			fb_readOut.m_Enable := FALSE;
			ton_wait_read_out.IN := FALSE;
			int_readOut := int_readOut +1;	
		ELSIF fb_readOut.fbMBRead_FC3.bError THEN
			fb_readOut.m_Enable := FALSE;
			ton_wait_read_out.IN := FALSE;
			int_readOut := int_readOut +1;		
		ELSIF ton_wait_read_out.Q THEN
			fb_readOut.m_Enable := FALSE;
			ton_wait_read_out.IN := FALSE;
			int_readOut := int_readOut +1;		
		END_IF			
	30: // wait state
		fb_readOut.m_Enable := FALSE;
		ton_wait_read_out.IN := TRUE;
		IF ton_wait_read_out.Q THEN
			ton_wait_read_out.IN := FALSE;
			int_readOut := int_readOut +1;
		END_IF			
	31: // read out IP 192.168.0.101 ID11  PV11 
		fb_readOut.m_Enable := TRUE;
		Str_Ip := '192.168.0.101';
		usint_ID := 11;
		int_Data_Received_old := fb_readout.int_Data_Received;
		int_readOut := int_readOut +1;
	32: // wait for received values	
		ton_wait_read_out.IN := TRUE;
		IF NOT fb_readOut.fbMBRead_FC3.bBusy AND int_Data_Received_old <> fb_readout.int_Data_Received  THEN
			y:=11;
			FOR z:=1 TO 20 BY 1 DO
				arrBuffer_FC3[y,z] := fb_readOut.w_Array_Received[z];
			END_FOR
			fb_readOut.m_Enable := FALSE;
			ton_wait_read_out.IN := FALSE;
			int_readOut := int_readOut +1;	
		ELSIF fb_readOut.fbMBRead_FC3.bError THEN
			fb_readOut.m_Enable := FALSE;
			ton_wait_read_out.IN := FALSE;
			int_readOut := int_readOut +1;		
		ELSIF ton_wait_read_out.Q THEN
			fb_readOut.m_Enable := FALSE;
			ton_wait_read_out.IN := FALSE;
			int_readOut := int_readOut +1;		
		END_IF			
	33: // wait state
		fb_readOut.m_Enable := FALSE;
		ton_wait_read_out.IN := TRUE;
		IF ton_wait_read_out.Q THEN
			ton_wait_read_out.IN := FALSE;
			int_readOut := int_readOut +1;
		END_IF			
	34: // read out IP 192.168.0.101 ID12  PV12 
		fb_readOut.m_Enable := TRUE;
		Str_Ip := '192.168.0.101';
		usint_ID := 12;
		int_Data_Received_old := fb_readout.int_Data_Received;
		int_readOut := int_readOut +1;
	35: // wait for received values	
		ton_wait_read_out.IN := TRUE;
		IF NOT fb_readOut.fbMBRead_FC3.bBusy AND int_Data_Received_old <> fb_readout.int_Data_Received  THEN
			y:=12;
			FOR z:=1 TO 20 BY 1 DO
				arrBuffer_FC3[y,z] := fb_readOut.w_Array_Received[z];
			END_FOR
			fb_readOut.m_Enable := FALSE;
			ton_wait_read_out.IN := FALSE;
			int_readOut := int_readOut +1;	
		ELSIF fb_readOut.fbMBRead_FC3.bError THEN
			fb_readOut.m_Enable := FALSE;
			ton_wait_read_out.IN := FALSE;
			int_readOut := int_readOut +1;		
		ELSIF ton_wait_read_out.Q THEN
			fb_readOut.m_Enable := FALSE;
			ton_wait_read_out.IN := FALSE;
			int_readOut := int_readOut +1;		
		END_IF			
	36: // wait state
		fb_readOut.m_Enable := FALSE;
		ton_wait_read_out.IN := TRUE;
		IF ton_wait_read_out.Q THEN
			ton_wait_read_out.IN := FALSE;
			int_readOut := int_readOut +1;
		END_IF			
	37: // read out IP 192.168.0.101 ID13  PV13 
		fb_readOut.m_Enable := TRUE;
		Str_Ip := '192.168.0.101';
		usint_ID := 13;
		int_Data_Received_old := fb_readout.int_Data_Received;
		int_readOut := int_readOut +1;
	38: // wait for received values	
		ton_wait_read_out.IN := TRUE;
		IF NOT fb_readOut.fbMBRead_FC3.bBusy AND int_Data_Received_old <> fb_readout.int_Data_Received  THEN
			y:=13;
			FOR z:=1 TO 20 BY 1 DO
				arrBuffer_FC3[y,z] := fb_readOut.w_Array_Received[z];
			END_FOR
			fb_readOut.m_Enable := FALSE;
			ton_wait_read_out.IN := FALSE;
			int_readOut := int_readOut +1;	
		ELSIF fb_readOut.fbMBRead_FC3.bError THEN
			fb_readOut.m_Enable := FALSE;
			ton_wait_read_out.IN := FALSE;
			int_readOut := int_readOut +1;		
		ELSIF ton_wait_read_out.Q THEN
			fb_readOut.m_Enable := FALSE;
			ton_wait_read_out.IN := FALSE;
			int_readOut := int_readOut +1;		
		END_IF			
	39: // wait state
		fb_readOut.m_Enable := FALSE;
		ton_wait_read_out.IN := TRUE;
		IF ton_wait_read_out.Q THEN
			ton_wait_read_out.IN := FALSE;
			int_readOut := int_readOut +1;
		END_IF			
	40: // read out IP 192.168.0.102 ID1  PV14 
		fb_readOut.m_Enable := TRUE;
		Str_Ip := '192.168.0.102';
		usint_ID := 1;
		int_Data_Received_old := fb_readout.int_Data_Received;
		int_readOut := int_readOut +1;
	41: // wait for received values	
		ton_wait_read_out.IN := TRUE;
		IF NOT fb_readOut.fbMBRead_FC3.bBusy AND int_Data_Received_old <> fb_readout.int_Data_Received  THEN
			y:=14;
			FOR z:=1 TO 20 BY 1 DO
				arrBuffer_FC3[y,z] := fb_readOut.w_Array_Received[z];
			END_FOR
			fb_readOut.m_Enable := FALSE;
			ton_wait_read_out.IN := FALSE;
			int_readOut := int_readOut +1;	
		ELSIF fb_readOut.fbMBRead_FC3.bError THEN
			fb_readOut.m_Enable := FALSE;
			ton_wait_read_out.IN := FALSE;
			int_readOut := int_readOut +1;		
		ELSIF ton_wait_read_out.Q THEN
			fb_readOut.m_Enable := FALSE;
			ton_wait_read_out.IN := FALSE;
			int_readOut := int_readOut +1;		
		END_IF			
	42: // wait state
		fb_readOut.m_Enable := FALSE;
		ton_wait_read_out.IN := TRUE;
		IF ton_wait_read_out.Q THEN
			ton_wait_read_out.IN := FALSE;
			int_readOut := int_readOut +1;
		END_IF
	43: // read out IP 192.168.0.103 ID1  PV15 
		fb_readOut.m_Enable := TRUE;
		Str_Ip := '192.168.0.103';
		usint_ID := 1;
		int_Data_Received_old := fb_readout.int_Data_Received;
		int_readOut := int_readOut +1;
	44: // wait for received values	
		ton_wait_read_out.IN := TRUE;
		IF NOT fb_readOut.fbMBRead_FC3.bBusy AND int_Data_Received_old <> fb_readout.int_Data_Received  THEN
			y:=14;
			FOR z:=1 TO 20 BY 1 DO
				arrBuffer_FC3[y,z] := fb_readOut.w_Array_Received[z];
			END_FOR
			fb_readOut.m_Enable := FALSE;
			ton_wait_read_out.IN := FALSE;
			int_readOut := int_readOut +1;	
		ELSIF fb_readOut.fbMBRead_FC3.bError THEN
			fb_readOut.m_Enable := FALSE;
			ton_wait_read_out.IN := FALSE;
			int_readOut := int_readOut +1;		
		ELSIF ton_wait_read_out.Q THEN
			fb_readOut.m_Enable := FALSE;
			ton_wait_read_out.IN := FALSE;
			int_readOut := int_readOut +1;		
		END_IF			
	45: // wait state
		fb_readOut.m_Enable := FALSE;
		ton_wait_read_out.IN := TRUE;
		IF ton_wait_read_out.Q THEN
			ton_wait_read_out.IN := FALSE;
			int_readOut := int_readOut +1;
		END_IF	

	46: // read out IP 192.168.0.104 ID1  PV16 
		fb_readOut.m_Enable := TRUE;
		Str_Ip := '192.168.0.104';
		usint_ID := 1;
		int_Data_Received_old := fb_readout.int_Data_Received;
		int_readOut := int_readOut +1;
	47: // wait for received values	
		ton_wait_read_out.IN := TRUE;
		IF NOT fb_readOut.fbMBRead_FC3.bBusy AND int_Data_Received_old <> fb_readout.int_Data_Received  THEN
			y:=16;
			FOR z:=1 TO 20 BY 1 DO
				arrBuffer_FC3[y,z] := fb_readOut.w_Array_Received[z];
			END_FOR
			fb_readOut.m_Enable := FALSE;
			ton_wait_read_out.IN := FALSE;
			int_readOut := int_readOut +1;	
		ELSIF fb_readOut.fbMBRead_FC3.bError THEN
			fb_readOut.m_Enable := FALSE;
			ton_wait_read_out.IN := FALSE;
			int_readOut := int_readOut +1;		
		ELSIF ton_wait_read_out.Q THEN
			fb_readOut.m_Enable := FALSE;
			ton_wait_read_out.IN := FALSE;
			int_readOut := int_readOut +1;		
		END_IF	
	48: // wait state
		fb_readOut.m_Enable := FALSE;
		ton_wait_read_out.IN := TRUE;
		IF ton_wait_read_out.Q THEN
			ton_wait_read_out.IN := FALSE;
			int_readOut := int_readOut +1;
		END_IF	
		
	49: // read out IP 192.168.0.104 ID2  PV17 
		fb_readOut.m_Enable := TRUE;
		Str_Ip := '192.168.0.104';
		usint_ID := 2;
		int_Data_Received_old := fb_readout.int_Data_Received;
		int_readOut := int_readOut +1;
	50: // wait for received values	
		ton_wait_read_out.IN := TRUE;
		IF NOT fb_readOut.fbMBRead_FC3.bBusy AND int_Data_Received_old <> fb_readout.int_Data_Received  THEN
			y:=17;
			FOR z:=1 TO 20 BY 1 DO
				arrBuffer_FC3[y,z] := fb_readOut.w_Array_Received[z];
			END_FOR
			fb_readOut.m_Enable := FALSE;
			ton_wait_read_out.IN := FALSE;
			int_readOut := int_readOut +1;	
		ELSIF fb_readOut.fbMBRead_FC3.bError THEN
			fb_readOut.m_Enable := FALSE;
			ton_wait_read_out.IN := FALSE;
			int_readOut := int_readOut +1;		
		ELSIF ton_wait_read_out.Q THEN
			fb_readOut.m_Enable := FALSE;
			ton_wait_read_out.IN := FALSE;
			int_readOut := int_readOut +1;		
		END_IF	
	51: // wait state
		fb_readOut.m_Enable := FALSE;
		ton_wait_read_out.IN := TRUE;
		IF ton_wait_read_out.Q THEN
			ton_wait_read_out.IN := FALSE;
			int_readOut := int_readOut +1;
		END_IF
		
		
	52: // read out IP 192.168.0.104 ID3  PV18 
		fb_readOut.m_Enable := TRUE;
		Str_Ip := '192.168.0.104';
		usint_ID := 3;
		int_Data_Received_old := fb_readout.int_Data_Received;
		int_readOut := int_readOut +1;
	53: // wait for received values	
		ton_wait_read_out.IN := TRUE;
		IF NOT fb_readOut.fbMBRead_FC3.bBusy AND int_Data_Received_old <> fb_readout.int_Data_Received  THEN
			y:=18;
			FOR z:=1 TO 20 BY 1 DO
				arrBuffer_FC3[y,z] := fb_readOut.w_Array_Received[z];
			END_FOR
			fb_readOut.m_Enable := FALSE;
			ton_wait_read_out.IN := FALSE;
			int_readOut := int_readOut +1;	
		ELSIF fb_readOut.fbMBRead_FC3.bError THEN
			fb_readOut.m_Enable := FALSE;
			ton_wait_read_out.IN := FALSE;
			int_readOut := int_readOut +1;		
		ELSIF ton_wait_read_out.Q THEN
			fb_readOut.m_Enable := FALSE;
			ton_wait_read_out.IN := FALSE;
			int_readOut := int_readOut +1;		
		END_IF	
	54: // wait state
		fb_readOut.m_Enable := FALSE;
		ton_wait_read_out.IN := TRUE;
		IF ton_wait_read_out.Q THEN
			ton_wait_read_out.IN := FALSE;
			int_readOut := int_readOut +1;
		END_IF
		
		
	55: // read out IP 192.168.0.104 ID4  PV19 
		fb_readOut.m_Enable := TRUE;
		Str_Ip := '192.168.0.104';
		usint_ID := 4;
		int_Data_Received_old := fb_readout.int_Data_Received;
		int_readOut := int_readOut +1;
	56: // wait for received values	
		ton_wait_read_out.IN := TRUE;
		IF NOT fb_readOut.fbMBRead_FC3.bBusy AND int_Data_Received_old <> fb_readout.int_Data_Received  THEN
			y:=19;
			FOR z:=1 TO 20 BY 1 DO
				arrBuffer_FC3[y,z] := fb_readOut.w_Array_Received[z];
			END_FOR
			fb_readOut.m_Enable := FALSE;
			ton_wait_read_out.IN := FALSE;
			int_readOut := int_readOut +1;	
		ELSIF fb_readOut.fbMBRead_FC3.bError THEN
			fb_readOut.m_Enable := FALSE;
			ton_wait_read_out.IN := FALSE;
			int_readOut := int_readOut +1;		
		ELSIF ton_wait_read_out.Q THEN
			fb_readOut.m_Enable := FALSE;
			ton_wait_read_out.IN := FALSE;
			int_readOut := int_readOut +1;		
		END_IF	
	57: // wait state
		fb_readOut.m_Enable := FALSE;
		ton_wait_read_out.IN := TRUE;
		IF ton_wait_read_out.Q THEN
			ton_wait_read_out.IN := FALSE;
			int_readOut := 60; //int_readOut +1;
		END_IF
		
		
	60:
		w:=1;		
		fbConvertWordToDword(wInputValue_1:= arrBuffer_FC3[w,3], wInputValue_2:= arrBuffer_FC3[w,4], eByteOrderForConvert:= eByteOrder.eBigEndian , dwOutputValue=> udint_Event1_PV1);
		fbConvertWordToDword(wInputValue_1:= arrBuffer_FC3[w,5], wInputValue_2:= arrBuffer_FC3[w,6], eByteOrderForConvert:= eByteOrder.eBigEndian , dwOutputValue=> udint_Event2_PV1);
		fbConvertWordToDword(wInputValue_1:= arrBuffer_FC3[w,7], wInputValue_2:= arrBuffer_FC3[w,8], eByteOrderForConvert:= eByteOrder.eBigEndian , dwOutputValue=> udint_VendorEvent1_PV1);
		fbConvertWordToDword(wInputValue_1:= arrBuffer_FC3[w,9], wInputValue_2:= arrBuffer_FC3[w,10], eByteOrderForConvert:= eByteOrder.eBigEndian , dwOutputValue=> udint_VendorEvent2_PV1);
		fbConvertWordToDword(wInputValue_1:= arrBuffer_FC3[w,11], wInputValue_2:= arrBuffer_FC3[w,12], eByteOrderForConvert:= eByteOrder.eBigEndian , dwOutputValue=> udint_VendorEvent3_PV1);
		w:=2;		
		fbConvertWordToDword(wInputValue_1:= arrBuffer_FC3[w,3], wInputValue_2:= arrBuffer_FC3[w,4], eByteOrderForConvert:= eByteOrder.eBigEndian , dwOutputValue=> udint_Event1_PV2);
		fbConvertWordToDword(wInputValue_1:= arrBuffer_FC3[w,5], wInputValue_2:= arrBuffer_FC3[w,6], eByteOrderForConvert:= eByteOrder.eBigEndian , dwOutputValue=> udint_Event2_PV2);
		fbConvertWordToDword(wInputValue_1:= arrBuffer_FC3[w,7], wInputValue_2:= arrBuffer_FC3[w,8], eByteOrderForConvert:= eByteOrder.eBigEndian , dwOutputValue=> udint_VendorEvent1_PV2);
		fbConvertWordToDword(wInputValue_1:= arrBuffer_FC3[w,9], wInputValue_2:= arrBuffer_FC3[w,10], eByteOrderForConvert:= eByteOrder.eBigEndian , dwOutputValue=> udint_VendorEvent2_PV2);
		fbConvertWordToDword(wInputValue_1:= arrBuffer_FC3[w,11], wInputValue_2:= arrBuffer_FC3[w,12], eByteOrderForConvert:= eByteOrder.eBigEndian , dwOutputValue=> udint_VendorEvent3_PV2);
		w:=3;		
		fbConvertWordToDword(wInputValue_1:= arrBuffer_FC3[w,3], wInputValue_2:= arrBuffer_FC3[w,4], eByteOrderForConvert:= eByteOrder.eBigEndian , dwOutputValue=> udint_Event1_PV3);
		fbConvertWordToDword(wInputValue_1:= arrBuffer_FC3[w,5], wInputValue_2:= arrBuffer_FC3[w,6], eByteOrderForConvert:= eByteOrder.eBigEndian , dwOutputValue=> udint_Event2_PV3);
		fbConvertWordToDword(wInputValue_1:= arrBuffer_FC3[w,7], wInputValue_2:= arrBuffer_FC3[w,8], eByteOrderForConvert:= eByteOrder.eBigEndian , dwOutputValue=> udint_VendorEvent1_PV3);
		fbConvertWordToDword(wInputValue_1:= arrBuffer_FC3[w,9], wInputValue_2:= arrBuffer_FC3[w,10], eByteOrderForConvert:= eByteOrder.eBigEndian , dwOutputValue=> udint_VendorEvent2_PV3);
		fbConvertWordToDword(wInputValue_1:= arrBuffer_FC3[w,11], wInputValue_2:= arrBuffer_FC3[w,12], eByteOrderForConvert:= eByteOrder.eBigEndian , dwOutputValue=> udint_VendorEvent3_PV3);
		w:=4;		
		fbConvertWordToDword(wInputValue_1:= arrBuffer_FC3[w,3], wInputValue_2:= arrBuffer_FC3[w,4], eByteOrderForConvert:= eByteOrder.eBigEndian , dwOutputValue=> udint_Event1_PV4);
		fbConvertWordToDword(wInputValue_1:= arrBuffer_FC3[w,5], wInputValue_2:= arrBuffer_FC3[w,6], eByteOrderForConvert:= eByteOrder.eBigEndian , dwOutputValue=> udint_Event2_PV4);
		fbConvertWordToDword(wInputValue_1:= arrBuffer_FC3[w,7], wInputValue_2:= arrBuffer_FC3[w,8], eByteOrderForConvert:= eByteOrder.eBigEndian , dwOutputValue=> udint_VendorEvent1_PV4);
		fbConvertWordToDword(wInputValue_1:= arrBuffer_FC3[w,9], wInputValue_2:= arrBuffer_FC3[w,10], eByteOrderForConvert:= eByteOrder.eBigEndian , dwOutputValue=> udint_VendorEvent2_PV4);
		fbConvertWordToDword(wInputValue_1:= arrBuffer_FC3[w,11], wInputValue_2:= arrBuffer_FC3[w,12], eByteOrderForConvert:= eByteOrder.eBigEndian , dwOutputValue=> udint_VendorEvent3_PV4);
		w:=5;		
		fbConvertWordToDword(wInputValue_1:= arrBuffer_FC3[w,3], wInputValue_2:= arrBuffer_FC3[w,4], eByteOrderForConvert:= eByteOrder.eBigEndian , dwOutputValue=> udint_Event1_PV5);
		fbConvertWordToDword(wInputValue_1:= arrBuffer_FC3[w,5], wInputValue_2:= arrBuffer_FC3[w,6], eByteOrderForConvert:= eByteOrder.eBigEndian , dwOutputValue=> udint_Event2_PV5);
		fbConvertWordToDword(wInputValue_1:= arrBuffer_FC3[w,7], wInputValue_2:= arrBuffer_FC3[w,8], eByteOrderForConvert:= eByteOrder.eBigEndian , dwOutputValue=> udint_VendorEvent1_PV5);
		fbConvertWordToDword(wInputValue_1:= arrBuffer_FC3[w,9], wInputValue_2:= arrBuffer_FC3[w,10], eByteOrderForConvert:= eByteOrder.eBigEndian , dwOutputValue=> udint_VendorEvent2_PV5);
		fbConvertWordToDword(wInputValue_1:= arrBuffer_FC3[w,11], wInputValue_2:= arrBuffer_FC3[w,12], eByteOrderForConvert:= eByteOrder.eBigEndian , dwOutputValue=> udint_VendorEvent3_PV5);
		w:=6;		
		fbConvertWordToDword(wInputValue_1:= arrBuffer_FC3[w,3], wInputValue_2:= arrBuffer_FC3[w,4], eByteOrderForConvert:= eByteOrder.eBigEndian , dwOutputValue=> udint_Event1_PV6);
		fbConvertWordToDword(wInputValue_1:= arrBuffer_FC3[w,5], wInputValue_2:= arrBuffer_FC3[w,6], eByteOrderForConvert:= eByteOrder.eBigEndian , dwOutputValue=> udint_Event2_PV6);
		fbConvertWordToDword(wInputValue_1:= arrBuffer_FC3[w,7], wInputValue_2:= arrBuffer_FC3[w,8], eByteOrderForConvert:= eByteOrder.eBigEndian , dwOutputValue=> udint_VendorEvent1_PV6);
		fbConvertWordToDword(wInputValue_1:= arrBuffer_FC3[w,9], wInputValue_2:= arrBuffer_FC3[w,10], eByteOrderForConvert:= eByteOrder.eBigEndian , dwOutputValue=> udint_VendorEvent2_PV6);
		fbConvertWordToDword(wInputValue_1:= arrBuffer_FC3[w,11], wInputValue_2:= arrBuffer_FC3[w,12], eByteOrderForConvert:= eByteOrder.eBigEndian , dwOutputValue=> udint_VendorEvent3_PV6);
		w:=7;		
		fbConvertWordToDword(wInputValue_1:= arrBuffer_FC3[w,3], wInputValue_2:= arrBuffer_FC3[w,4], eByteOrderForConvert:= eByteOrder.eBigEndian , dwOutputValue=> udint_Event1_PV7);
		fbConvertWordToDword(wInputValue_1:= arrBuffer_FC3[w,5], wInputValue_2:= arrBuffer_FC3[w,6], eByteOrderForConvert:= eByteOrder.eBigEndian , dwOutputValue=> udint_Event2_PV7);
		fbConvertWordToDword(wInputValue_1:= arrBuffer_FC3[w,7], wInputValue_2:= arrBuffer_FC3[w,8], eByteOrderForConvert:= eByteOrder.eBigEndian , dwOutputValue=> udint_VendorEvent1_PV7);
		fbConvertWordToDword(wInputValue_1:= arrBuffer_FC3[w,9], wInputValue_2:= arrBuffer_FC3[w,10], eByteOrderForConvert:= eByteOrder.eBigEndian , dwOutputValue=> udint_VendorEvent2_PV7);
		fbConvertWordToDword(wInputValue_1:= arrBuffer_FC3[w,11], wInputValue_2:= arrBuffer_FC3[w,12], eByteOrderForConvert:= eByteOrder.eBigEndian , dwOutputValue=> udint_VendorEvent3_PV7);
		w:=8;		
		fbConvertWordToDword(wInputValue_1:= arrBuffer_FC3[w,3], wInputValue_2:= arrBuffer_FC3[w,4], eByteOrderForConvert:= eByteOrder.eBigEndian , dwOutputValue=> udint_Event1_PV8);
		fbConvertWordToDword(wInputValue_1:= arrBuffer_FC3[w,5], wInputValue_2:= arrBuffer_FC3[w,6], eByteOrderForConvert:= eByteOrder.eBigEndian , dwOutputValue=> udint_Event2_PV8);
		fbConvertWordToDword(wInputValue_1:= arrBuffer_FC3[w,7], wInputValue_2:= arrBuffer_FC3[w,8], eByteOrderForConvert:= eByteOrder.eBigEndian , dwOutputValue=> udint_VendorEvent1_PV8);
		fbConvertWordToDword(wInputValue_1:= arrBuffer_FC3[w,9], wInputValue_2:= arrBuffer_FC3[w,10], eByteOrderForConvert:= eByteOrder.eBigEndian , dwOutputValue=> udint_VendorEvent2_PV8);
		fbConvertWordToDword(wInputValue_1:= arrBuffer_FC3[w,11], wInputValue_2:= arrBuffer_FC3[w,12], eByteOrderForConvert:= eByteOrder.eBigEndian , dwOutputValue=> udint_VendorEvent3_PV8);
		w:=9;		
		fbConvertWordToDword(wInputValue_1:= arrBuffer_FC3[w,3], wInputValue_2:= arrBuffer_FC3[w,4], eByteOrderForConvert:= eByteOrder.eBigEndian , dwOutputValue=> udint_Event1_PV9);
		fbConvertWordToDword(wInputValue_1:= arrBuffer_FC3[w,5], wInputValue_2:= arrBuffer_FC3[w,6], eByteOrderForConvert:= eByteOrder.eBigEndian , dwOutputValue=> udint_Event2_PV9);
		fbConvertWordToDword(wInputValue_1:= arrBuffer_FC3[w,7], wInputValue_2:= arrBuffer_FC3[w,8], eByteOrderForConvert:= eByteOrder.eBigEndian , dwOutputValue=> udint_VendorEvent1_PV9);
		fbConvertWordToDword(wInputValue_1:= arrBuffer_FC3[w,9], wInputValue_2:= arrBuffer_FC3[w,10], eByteOrderForConvert:= eByteOrder.eBigEndian , dwOutputValue=> udint_VendorEvent2_PV9);
		fbConvertWordToDword(wInputValue_1:= arrBuffer_FC3[w,11], wInputValue_2:= arrBuffer_FC3[w,12], eByteOrderForConvert:= eByteOrder.eBigEndian , dwOutputValue=> udint_VendorEvent3_PV9);
		w:=10;		
		fbConvertWordToDword(wInputValue_1:= arrBuffer_FC3[w,3], wInputValue_2:= arrBuffer_FC3[w,4], eByteOrderForConvert:= eByteOrder.eBigEndian , dwOutputValue=> udint_Event1_PV10);
		fbConvertWordToDword(wInputValue_1:= arrBuffer_FC3[w,5], wInputValue_2:= arrBuffer_FC3[w,6], eByteOrderForConvert:= eByteOrder.eBigEndian , dwOutputValue=> udint_Event2_PV10);
		fbConvertWordToDword(wInputValue_1:= arrBuffer_FC3[w,7], wInputValue_2:= arrBuffer_FC3[w,8], eByteOrderForConvert:= eByteOrder.eBigEndian , dwOutputValue=> udint_VendorEvent1_PV10);
		fbConvertWordToDword(wInputValue_1:= arrBuffer_FC3[w,9], wInputValue_2:= arrBuffer_FC3[w,10], eByteOrderForConvert:= eByteOrder.eBigEndian , dwOutputValue=> udint_VendorEvent2_PV10);
		fbConvertWordToDword(wInputValue_1:= arrBuffer_FC3[w,11], wInputValue_2:= arrBuffer_FC3[w,12], eByteOrderForConvert:= eByteOrder.eBigEndian , dwOutputValue=> udint_VendorEvent3_PV10);
		w:=11;		
		fbConvertWordToDword(wInputValue_1:= arrBuffer_FC3[w,3], wInputValue_2:= arrBuffer_FC3[w,4], eByteOrderForConvert:= eByteOrder.eBigEndian , dwOutputValue=> udint_Event1_PV11);
		fbConvertWordToDword(wInputValue_1:= arrBuffer_FC3[w,5], wInputValue_2:= arrBuffer_FC3[w,6], eByteOrderForConvert:= eByteOrder.eBigEndian , dwOutputValue=> udint_Event2_PV11);
		fbConvertWordToDword(wInputValue_1:= arrBuffer_FC3[w,7], wInputValue_2:= arrBuffer_FC3[w,8], eByteOrderForConvert:= eByteOrder.eBigEndian , dwOutputValue=> udint_VendorEvent1_PV11);
		fbConvertWordToDword(wInputValue_1:= arrBuffer_FC3[w,9], wInputValue_2:= arrBuffer_FC3[w,10], eByteOrderForConvert:= eByteOrder.eBigEndian , dwOutputValue=> udint_VendorEvent2_PV11);
		fbConvertWordToDword(wInputValue_1:= arrBuffer_FC3[w,11], wInputValue_2:= arrBuffer_FC3[w,12], eByteOrderForConvert:= eByteOrder.eBigEndian , dwOutputValue=> udint_VendorEvent3_PV11);
		w:=12;		
		fbConvertWordToDword(wInputValue_1:= arrBuffer_FC3[w,3], wInputValue_2:= arrBuffer_FC3[w,4], eByteOrderForConvert:= eByteOrder.eBigEndian , dwOutputValue=> udint_Event1_PV12);
		fbConvertWordToDword(wInputValue_1:= arrBuffer_FC3[w,5], wInputValue_2:= arrBuffer_FC3[w,6], eByteOrderForConvert:= eByteOrder.eBigEndian , dwOutputValue=> udint_Event2_PV12);
		fbConvertWordToDword(wInputValue_1:= arrBuffer_FC3[w,7], wInputValue_2:= arrBuffer_FC3[w,8], eByteOrderForConvert:= eByteOrder.eBigEndian , dwOutputValue=> udint_VendorEvent1_PV12);
		fbConvertWordToDword(wInputValue_1:= arrBuffer_FC3[w,9], wInputValue_2:= arrBuffer_FC3[w,10], eByteOrderForConvert:= eByteOrder.eBigEndian , dwOutputValue=> udint_VendorEvent2_PV12);
		fbConvertWordToDword(wInputValue_1:= arrBuffer_FC3[w,11], wInputValue_2:= arrBuffer_FC3[w,12], eByteOrderForConvert:= eByteOrder.eBigEndian , dwOutputValue=> udint_VendorEvent3_PV12);
		w:=13;		
		fbConvertWordToDword(wInputValue_1:= arrBuffer_FC3[w,3], wInputValue_2:= arrBuffer_FC3[w,4], eByteOrderForConvert:= eByteOrder.eBigEndian , dwOutputValue=> udint_Event1_PV13);
		fbConvertWordToDword(wInputValue_1:= arrBuffer_FC3[w,5], wInputValue_2:= arrBuffer_FC3[w,6], eByteOrderForConvert:= eByteOrder.eBigEndian , dwOutputValue=> udint_Event2_PV13);
		fbConvertWordToDword(wInputValue_1:= arrBuffer_FC3[w,7], wInputValue_2:= arrBuffer_FC3[w,8], eByteOrderForConvert:= eByteOrder.eBigEndian , dwOutputValue=> udint_VendorEvent1_PV13);
		fbConvertWordToDword(wInputValue_1:= arrBuffer_FC3[w,9], wInputValue_2:= arrBuffer_FC3[w,10], eByteOrderForConvert:= eByteOrder.eBigEndian , dwOutputValue=> udint_VendorEvent2_PV13);
		fbConvertWordToDword(wInputValue_1:= arrBuffer_FC3[w,11], wInputValue_2:= arrBuffer_FC3[w,12], eByteOrderForConvert:= eByteOrder.eBigEndian , dwOutputValue=> udint_VendorEvent3_PV13);
		w:=14;		
		fbConvertWordToDword(wInputValue_1:= arrBuffer_FC3[w,3], wInputValue_2:= arrBuffer_FC3[w,4], eByteOrderForConvert:= eByteOrder.eBigEndian , dwOutputValue=> udint_Event1_PV14);
		fbConvertWordToDword(wInputValue_1:= arrBuffer_FC3[w,5], wInputValue_2:= arrBuffer_FC3[w,6], eByteOrderForConvert:= eByteOrder.eBigEndian , dwOutputValue=> udint_Event2_PV14);
		fbConvertWordToDword(wInputValue_1:= arrBuffer_FC3[w,7], wInputValue_2:= arrBuffer_FC3[w,8], eByteOrderForConvert:= eByteOrder.eBigEndian , dwOutputValue=> udint_VendorEvent1_PV14);
		fbConvertWordToDword(wInputValue_1:= arrBuffer_FC3[w,9], wInputValue_2:= arrBuffer_FC3[w,10], eByteOrderForConvert:= eByteOrder.eBigEndian , dwOutputValue=> udint_VendorEvent2_PV14);
		fbConvertWordToDword(wInputValue_1:= arrBuffer_FC3[w,11], wInputValue_2:= arrBuffer_FC3[w,12], eByteOrderForConvert:= eByteOrder.eBigEndian , dwOutputValue=> udint_VendorEvent3_PV14);
		w:=15;		
		fbConvertWordToDword(wInputValue_1:= arrBuffer_FC3[w,3], wInputValue_2:= arrBuffer_FC3[w,4], eByteOrderForConvert:= eByteOrder.eBigEndian , dwOutputValue=> udint_Event1_PV15);
		fbConvertWordToDword(wInputValue_1:= arrBuffer_FC3[w,5], wInputValue_2:= arrBuffer_FC3[w,6], eByteOrderForConvert:= eByteOrder.eBigEndian , dwOutputValue=> udint_Event2_PV15);
		fbConvertWordToDword(wInputValue_1:= arrBuffer_FC3[w,7], wInputValue_2:= arrBuffer_FC3[w,8], eByteOrderForConvert:= eByteOrder.eBigEndian , dwOutputValue=> udint_VendorEvent1_PV15);
		fbConvertWordToDword(wInputValue_1:= arrBuffer_FC3[w,9], wInputValue_2:= arrBuffer_FC3[w,10], eByteOrderForConvert:= eByteOrder.eBigEndian , dwOutputValue=> udint_VendorEvent2_PV15);
		fbConvertWordToDword(wInputValue_1:= arrBuffer_FC3[w,11], wInputValue_2:= arrBuffer_FC3[w,12], eByteOrderForConvert:= eByteOrder.eBigEndian , dwOutputValue=> udint_VendorEvent3_PV15);
		w:=16;		
		fbConvertWordToDword(wInputValue_1:= arrBuffer_FC3[w,3], wInputValue_2:= arrBuffer_FC3[w,4], eByteOrderForConvert:= eByteOrder.eBigEndian , dwOutputValue=> udint_Event1_PV16);
		fbConvertWordToDword(wInputValue_1:= arrBuffer_FC3[w,5], wInputValue_2:= arrBuffer_FC3[w,6], eByteOrderForConvert:= eByteOrder.eBigEndian , dwOutputValue=> udint_Event2_PV16);
		fbConvertWordToDword(wInputValue_1:= arrBuffer_FC3[w,7], wInputValue_2:= arrBuffer_FC3[w,8], eByteOrderForConvert:= eByteOrder.eBigEndian , dwOutputValue=> udint_VendorEvent1_PV16);
		fbConvertWordToDword(wInputValue_1:= arrBuffer_FC3[w,9], wInputValue_2:= arrBuffer_FC3[w,10], eByteOrderForConvert:= eByteOrder.eBigEndian , dwOutputValue=> udint_VendorEvent2_PV16);
		fbConvertWordToDword(wInputValue_1:= arrBuffer_FC3[w,11], wInputValue_2:= arrBuffer_FC3[w,12], eByteOrderForConvert:= eByteOrder.eBigEndian , dwOutputValue=> udint_VendorEvent3_PV16);
		w:=17;		
		fbConvertWordToDword(wInputValue_1:= arrBuffer_FC3[w,3], wInputValue_2:= arrBuffer_FC3[w,4], eByteOrderForConvert:= eByteOrder.eBigEndian , dwOutputValue=> udint_Event1_PV17);
		fbConvertWordToDword(wInputValue_1:= arrBuffer_FC3[w,5], wInputValue_2:= arrBuffer_FC3[w,6], eByteOrderForConvert:= eByteOrder.eBigEndian , dwOutputValue=> udint_Event2_PV17);
		fbConvertWordToDword(wInputValue_1:= arrBuffer_FC3[w,7], wInputValue_2:= arrBuffer_FC3[w,8], eByteOrderForConvert:= eByteOrder.eBigEndian , dwOutputValue=> udint_VendorEvent1_PV17);
		fbConvertWordToDword(wInputValue_1:= arrBuffer_FC3[w,9], wInputValue_2:= arrBuffer_FC3[w,10], eByteOrderForConvert:= eByteOrder.eBigEndian , dwOutputValue=> udint_VendorEvent2_PV17);
		fbConvertWordToDword(wInputValue_1:= arrBuffer_FC3[w,11], wInputValue_2:= arrBuffer_FC3[w,12], eByteOrderForConvert:= eByteOrder.eBigEndian , dwOutputValue=> udint_VendorEvent3_PV17);
		w:=18;		
		fbConvertWordToDword(wInputValue_1:= arrBuffer_FC3[w,3], wInputValue_2:= arrBuffer_FC3[w,4], eByteOrderForConvert:= eByteOrder.eBigEndian , dwOutputValue=> udint_Event1_PV18);
		fbConvertWordToDword(wInputValue_1:= arrBuffer_FC3[w,5], wInputValue_2:= arrBuffer_FC3[w,6], eByteOrderForConvert:= eByteOrder.eBigEndian , dwOutputValue=> udint_Event2_PV18);
		fbConvertWordToDword(wInputValue_1:= arrBuffer_FC3[w,7], wInputValue_2:= arrBuffer_FC3[w,8], eByteOrderForConvert:= eByteOrder.eBigEndian , dwOutputValue=> udint_VendorEvent1_PV18);
		fbConvertWordToDword(wInputValue_1:= arrBuffer_FC3[w,9], wInputValue_2:= arrBuffer_FC3[w,10], eByteOrderForConvert:= eByteOrder.eBigEndian , dwOutputValue=> udint_VendorEvent2_PV18);
		fbConvertWordToDword(wInputValue_1:= arrBuffer_FC3[w,11], wInputValue_2:= arrBuffer_FC3[w,12], eByteOrderForConvert:= eByteOrder.eBigEndian , dwOutputValue=> udint_VendorEvent3_PV18);
		w:=19;		
		fbConvertWordToDword(wInputValue_1:= arrBuffer_FC3[w,3], wInputValue_2:= arrBuffer_FC3[w,4], eByteOrderForConvert:= eByteOrder.eBigEndian , dwOutputValue=> udint_Event1_PV19);
		fbConvertWordToDword(wInputValue_1:= arrBuffer_FC3[w,5], wInputValue_2:= arrBuffer_FC3[w,6], eByteOrderForConvert:= eByteOrder.eBigEndian , dwOutputValue=> udint_Event2_PV19);
		fbConvertWordToDword(wInputValue_1:= arrBuffer_FC3[w,7], wInputValue_2:= arrBuffer_FC3[w,8], eByteOrderForConvert:= eByteOrder.eBigEndian , dwOutputValue=> udint_VendorEvent1_PV19);
		fbConvertWordToDword(wInputValue_1:= arrBuffer_FC3[w,9], wInputValue_2:= arrBuffer_FC3[w,10], eByteOrderForConvert:= eByteOrder.eBigEndian , dwOutputValue=> udint_VendorEvent2_PV19);
		fbConvertWordToDword(wInputValue_1:= arrBuffer_FC3[w,11], wInputValue_2:= arrBuffer_FC3[w,12], eByteOrderForConvert:= eByteOrder.eBigEndian , dwOutputValue=> udint_VendorEvent3_PV19);
	
		int_readOut := 0;		
END_CASE

// test
fbConvertWordToDword(wInputValue_1:= word_1, wInputValue_2:= word_2, eByteOrderForConvert:= eByteOrder.eBigEndian , dwOutputValue=> udint_Out);



ton_wait_read_out( 	In :=,
					PT := T#1S);
	
fb_readOut(
	m_Enable:= , 
	str_IPAdress:=Str_Ip , 
	w_Adress:=w_Adress , 
	usint_Quantity:= usint_Quantity, 
	usint_ID:= usint_ID,
	m_PollSuccessful=> , 
	w_Array_Received=> , 
	udint_Error_ID=> );
	
// Modbus Fault for each PV 
	
b_ModbusFault_PV_1 :=  	fbPV.arrDataSymo10[1].eErrorState = 1;
b_ModbusFault_PV_2 :=  	fbPV.arrDataSymo10[2].eErrorState = 1;
b_ModbusFault_PV_3 :=  	fbPV.arrDataSymo10[3].eErrorState = 1;
b_ModbusFault_PV_4 :=  	fbPV.arrDataSymo10[4].eErrorState = 1;
b_ModbusFault_PV_5 :=  	fbPV.arrDataSymo10[5].eErrorState = 1;
b_ModbusFault_PV_6 :=  	fbPV.arrDataSymo10[6].eErrorState = 1;
b_ModbusFault_PV_7 :=  	fbPV.arrDataSymo10[7].eErrorState = 1;
b_ModbusFault_PV_8 :=  	fbPV.arrDataSymo10[8].eErrorState = 1;
b_ModbusFault_PV_9 :=  	fbPV.arrDataSymo10[9].eErrorState = 1;
b_ModbusFault_PV_10:=  	fbPV.arrDataSymo10[10].eErrorState = 1;
b_ModbusFault_PV_11:=  	fbPV.arrDataSymo10[11].eErrorState = 1;
b_ModbusFault_PV_12:=  	fbPV.arrDataSymo10[12].eErrorState = 1;
b_ModbusFault_PV_13:=  	fbPV.arrDataSymo10[13].eErrorState = 1;
b_ModbusFault_PV_14:=  	fbPV_2.arrDataSymo10[1].eErrorState = 1;
b_ModbusFault_PV_15 :=  fbPV_3.arrDataSymo10[1].eErrorState = 1;
b_ModbusFault_PV_16 :=  fbPV_4.arrDataSymo10[1].eErrorState = 1;
b_ModbusFault_PV_17 :=  fbPV_4.arrDataSymo10[2].eErrorState = 1;
b_ModbusFault_PV_18 :=  fbPV_4.arrDataSymo10[3].eErrorState = 1;
b_ModbusFault_PV_19 :=  fbPV_4.arrDataSymo10[4].eErrorState = 1;

b_ModbusFault_PV_any := b_ModbusFault_PV_1 OR b_ModbusFault_PV_2 OR b_ModbusFault_PV_3 OR b_ModbusFault_PV_4 OR b_ModbusFault_PV_5 OR b_ModbusFault_PV_6
						 OR b_ModbusFault_PV_7 OR b_ModbusFault_PV_8 OR b_ModbusFault_PV_9 OR b_ModbusFault_PV_10 OR b_ModbusFault_PV_11 OR b_ModbusFault_PV_12;

END_PROGRAM

// ---- FB/FB_ModBus_100Registers_FC3_inclID.TcPOU
FUNCTION_BLOCK FB_ModBus_100Registers_FC3_inclID
VAR_INPUT PERSISTENT
	m_Enable					: BOOL;						//Enable the Fuctionblock and his logic
	str_IPAdress				: STRING(15);				//IP Adress of the meter
	w_Adress					: WORD;						//modbus adress
	usint_Quantity				: usINT;						//Number of Words to get polled, max 100
	usint_ID					: USINT;						//Number of Words to get polled, max 100
END_VAR
VAR_OUTPUT
	m_PollSuccessful			: BOOL;						//Poll succesfull		
	w_Array_Received			: ARRAY[1..100] OF WORD;	// received data
	udint_Error_ID				: UDINT;					// ERR ID FB_MBReadRegs
END_VAR
VAR
	
	timer_Delay					: TON;						//Timer for Delay between Requests
	
	timer_DelayStart			: TON;						//Timer to start the state machine with Delay after enabling or after the system ist restartet
	
	timer_TimeOut				: TON;						//Timer for Timeout MB Read
	
	iStateModbusRead			: INT;						//State machine for read out Data over Modbus RTU
	
	fbMBRead_FC3				: FB_MBReadRegs  ;		//Modbus Read Function (FC3)
	
	ftrig_PEnable				: f_trig;					//Internal positive Edge
	
	iStateModbusError			: INT;						//State machine for error out Data over Modbus TCP/IP	
	
	FPError_FC_3				: R_TRIG;					//Internal positive Edge
	
	arrBuffer_FC3				: ARRAY[1..100] OF WORD;		//Buffer with Data from FC3
	
	timer_Connection_ok			: TON;
	int_Data_Received			: INT;
	
	m_MBTCPError				: BOOL;
	
	int_Data_Received_old		: INT;
	
	timer_Connection_ok_TOF	: TOF;
	
	fbConvertWordToDword		: FB_CV_WORD_TO_DWORD;			//Convert Word to Dword
	
	m_Poll_ok: BOOL;
	
	timer_Wait: Ton;
	int_TimeoutError: INT;
	int_FC3Error: INT;

END_VAR

(*	{attribute 'hide'}--------------------------------------------------------------------------------------------Limits-------------------------------------------------------------------------------------*)

w_Adress := LIMIT(0,w_Adress,60000);
usint_Quantity := LIMIT(1,usint_Quantity,100);
	
(*--------------------------------------------------------------------------------------------State Machine Read--------------------------------------------------------------------------------------*)

//Timer for Delay
timer_Delay(IN:= , PT:= T#50MS, Q=> , ET=> );

//Timeout Timer is dissabled when the Init Step is aktiv or the function is not enabled
IF iStateModbusRead = 0 OR NOT m_Enable THEN 
	timer_Timeout.IN := FALSE; 
END_IF
timer_Timeout(IN:= , PT:= T#1S, Q=> , ET=> );

//Enable with Delay that not all sockets have to be created at the same time
timer_DelayStart(IN:= m_Enable, PT:= T#1S, Q=> , ET=> );
ftrig_PEnable(CLK:= timer_DelayStart.Q, Q=> );

IF ftrig_PEnable.Q AND iStateModbusRead = 0 THEN 
	iStateModbusRead := 1; 
END_IF		
IF usint_ID < 1 OR usint_ID >255 THEN 
	usint_ID := 1;
END_IF		
//Not Enabled
IF NOT m_Enable THEN 
	iStateModbusRead := 0; 
	iStateModbusError := 0; 
END_IF		
		
CASE iStateModbusRead OF

	0://Init Step 
		timer_Delay.IN := FALSE;
		fbMBRead_FC3.bExecute := FALSE;
		m_Poll_ok:=FALSE;
		int_Data_Received:=0;
	
		iStateModbusRead := 1;
	
	1://read the required registers
		//Start Read
		fbMBRead_FC3.nQuantity := usint_Quantity;
		fbMBRead_FC3.nMBAddr := w_Adress;
		fbMBRead_FC3.bExecute := TRUE;
		fbMBRead_FC3.nUnitID := usint_ID;
		timer_Timeout.IN := TRUE;
		IF fbMBRead_FC3.bBusy THEN 
			timer_Delay.IN := TRUE; 
		END_IF
		
		//Wait for Delay, copy Data and then next step
		IF NOT fbMBRead_FC3.bBusy AND NOT fbMBRead_FC3.bError AND timer_Delay.Q THEN
			m_Poll_ok:=TRUE;
			int_Data_Received:=int_Data_Received+1;
			m_MBTCPError := FALSE; 
			
			w_Array_Received := arrBuffer_FC3;
			
			
			//Go to Next Step
			timer_Timeout.IN := FALSE;
			fbMBRead_FC3.bExecute := FALSE;
			timer_Delay.IN := FALSE;		
			iStateModbusRead := 3;
		END_IF	

		//Error or Timeout
		IF FPError_FC_3.Q THEN 
			iStateModbusError := 300;
			int_FC3Error := int_FC3Error+1;
		ELSIF timer_Timeout.Q THEN  
			timer_Timeout.IN := FALSE; 	
			iStateModbusError := 300;
			int_TimeoutError := int_TimeoutError+1;
		END_IF
		
	
	3://Wait and go to step 1
		//1 because 0 is the Init Step for Read
		timer_Wait.IN := TRUE;
		
		IF timer_Wait.Q = TRUE THEN
			iStateModbusRead := 1;
			timer_Wait.IN :=FALSE;
		END_IF

			
		
		//Error on Master, changes on Inputs or Timeout
		IF timer_Timeout.Q THEN 
			iStateModbusError := 300; 
		END_IF
	
END_CASE

(* wait timer*)

timer_Wait(PT:=T#3S);


(*------------------------------------------------------------------Error and Warning----------------------------------------------------------------------------*)	
 
timer_Connection_ok			(In:=int_Data_Received<>int_Data_Received_old,PT:=T#10S);
timer_Connection_ok_TOF		(In:=NOT(int_Data_Received<>int_Data_Received_old) AND int_Data_Received>3 ,PT:=T#20S);
int_Data_Received_old:=int_Data_Received;
m_PollSuccessful:=NOT timer_Connection_ok.Q AND timer_Connection_ok_TOF.Q ;

(*------------------------------------------------------------------------------------------Modbus TCP Functions---------------------------------------------------------------------------------------------*)

fbMBRead_FC3(	sIPAddr:= str_IPAdress, 
				nTCPPort:= 502,
				cbLength:= SIZEOF(arrBuffer_FC3), 
				pDestAddr:= ADR(arrBuffer_FC3), 
				tTimeout:= T#10S,
				nErrId => udint_Error_ID);

FPError_FC_3(CLK:= fbMBRead_FC3.bError, Q=> );		

(*------------------------------------------------------------------------------------------State Machine Error---------------------------------------------------------------------------------------------*)	

CASE iStateModbusError OF
	
	300://Error
		timer_Wait.IN :=TRUE;
		timer_Delay.IN := FALSE;
		fbMBRead_FC3.bExecute := FALSE;
		m_MBTCPError := TRUE; 		
		m_Poll_ok:=FALSE;
		int_Data_Received:=0;
				//Restart from new with the Read out part after an Error
		IF timer_Wait.Q = TRUE THEN
			iStateModbusRead := 0;	
			iStateModbusError := 0;
			timer_Wait.IN :=FALSE;
			timer_Timeout.IN := FALSE;
		END_IF		
							
END_CASE

END_FUNCTION_BLOCK

// ---- POUs/prgBattery.TcPOU
PROGRAM prgBattery
VAR PERSISTENT
	bEnableBattery				: BOOL;							//{#lynus.ag#()}
	byPrioBattery				: BYTE;							//{#lynus.ag#()}
	lrMaxCapacityBattery		: LREAL;						//{#lynus.ag#()}
	lrCounterBattProd			: LREAL;						//{#lynus.ag#()}
	lrCounterBattCons			: LREAL;						//{#lynus.ag#()}
	by_Min_BatterySOC			: BYTE;							//{#lynus.ag#()}
	by_Max_BatterySOC			: BYTE;							//{#lynus.ag#()}
END_VAR
VAR
	fbBattery					: FB_Xelectrix_Powerbox_v2_2;
	fbBattCounter				: FB_EnergyCounter;
	bIsEnabledBattery			: BOOL;							//{#lynus.ag#()}
	bResetBattery				: BOOL;							//{#lynus.ag#()}
	bSResetBattery				: BOOL;							//{#lynus.ag#()}
	byErrorWarningBattery		: BYTE;							//{#lynus.ag#()}
	dwSOCBattery				: DWORD;						//{#lynus.ag#()}
	rTargetPowerBattery			: REAL;							//{#lynus.ag#()}
	lrPowerBattery				: LREAL;						//{#lynus.ag#()}
	lrActualCapacityBattery		: LREAL;						//{#lynus.ag#()}
	mtest: BOOL;
	x:INT;

	int_GridState: INT;											//{#lynus.ag#()}
	int_BatteryState: INT;										//{#lynus.ag#()}
	int_OperatingState: INT;									//{#lynus.ag#()}
	int_ErrorState: INT;										//{#lynus.ag#()}

	FB_Interval: FB_IntervalBit;
	m_IslandOperationStart: BOOL;								//{#lynus.ag#()}
	m_IslandOperationOngoing: BOOL;								//{#lynus.ag#()}
	m_IslandOperationStop: BOOL;								//{#lynus.ag#()}
	t_Interval :TIME:=T#60M;
	t_HightTime :TIME:=T#1S;
	
	m_BatteryErrorActive: BOOL;									//{#lynus.ag#()}
	m_BatteryModbusCommError: BOOL;								//{#lynus.ag#()}
	m_BatteryTargetSPError: BOOL;								//{#lynus.ag#()}
	Ton_Delay_BatteryError: Ton;
	Ton_Delay_BatteryModbusError: Ton;
	Ton_Delay_BatterySPError: Ton;	
	b_Battery_ModbusFault		: BOOL;							//{#lynus.ag#()}
	by_S_Min_BatterySOC			: BYTE;							//{#lynus.ag#()}
	by_S_Max_BatterySOC			: BYTE;							//{#lynus.ag#()}

END_VAR

IF mtest THEN
	Lynus_Standards.GVL_Energy.stDataOfBatteryInverters[1,1].rTargetPowerEMS:=x;
 END_IF

fbBattery(
	bEnable:= bEnableBattery, 
	bActivateControl:= TRUE, 
	byUnitID:= 1, 
	byPriority:= byPrioBattery, 
	diNrOfEMS_IN:= prgEMS.fbEMS.diNrOfEMS_OUT, 
	lrMaxCapacityBattery:= lrMaxCapacityBattery, 
	sIPAdress:= '10.11.90.120',   //192.168.0.110',
	bReset:= bResetBattery, 
	by_minDischargeSOC := by_Min_BatterySOC,
	by_maxChargeSOC := by_Max_BatterySOC,
	stDataXelectrix=> , 
	stDataBatt=> , 
	stDataBattInverter=> , 
	stDataEMPower_Grid=> , 
	stDataEMCounter_Grid=> , 
	diNrOfBatt_OUT=> , 
	diNrOfBattInverter_OUT=> , 
	diNrOfEM_OUT_Grid=> , 
	lrMaxCapacityBattery_OUT=> ,
	by_SminDischargeSOC	=> by_S_Min_BatterySOC,	
	by_SmaxChargeSOC=> by_S_Max_BatterySOC
);
	
//Out
bIsEnabledBattery := fbBattery.stDataBatt.bEnabled;
	bSResetBattery := fbBattery.stDataBattInverter.bStateReset;
		dwSOCBattery := fbBattery.stDataBatt.dwSOC;
			rTargetPowerBattery := fbBattery.stDataBattInverter.rTargetPower;
				lrPowerBattery := fbBattery.stDataBatt.lrPower;
					lrActualCapacityBattery := fbBattery.stDataBatt.lrCapacity;
						byErrorWarningBattery := fbBattery.stDataBatt.byErrorWarning;
							

// EnergyCounter
fbBattCounter(
	byActiveTariff:= 1, 
	lrPowerInput:= lrPowerBattery, 
	lrTotalCounterEnergy_Consumption=> , 
	lrTotalCounterEnergy_Production=> , 
	lrCounterEnergyT1_Consumption=> , 
	lrCounterEnergyT2_Consumption=> , 
	lrCounterEnergyT1_Production=> , 
	lrCounterEnergyT2_Production=> );
	
IF fbBattCounter.lrTotalCounterEnergy_Production > lrCounterBattProd THEN  	
	lrCounterBattProd := fbBattCounter.lrTotalCounterEnergy_Production;
END_IF

IF fbBattCounter.lrTotalCounterEnergy_Consumption > lrCounterBattCons THEN  	
	lrCounterBattCons := fbBattCounter.lrTotalCounterEnergy_Consumption;
END_IF

// send e states to cloud
int_GridState 		:= fbBattery.stDataXelectrix.eGridState;
int_BatteryState	:= fbBattery.stDataXelectrix.eBatteryState;
int_OperatingState	:= fbBattery.stDataXelectrix.eOperatingState;
int_ErrorState		:= fbBattery.stDataXelectrix.eErrorState;


// create bits when battery is in island operation

FB_Interval(
	m_Input			:=  prgBattery.fbBattery.stDataXelectrix.eGridState = 2,	//   2 = Island Mode 
	t_Interval 		:= t_Interval , 
	t_HighTime		:= t_HightTime, 
	m_RisingEdge	=> m_IslandOperationStart, 
	m_Interval		=> m_IslandOperationOngoing, 
	m_FallingEdge	=> m_IslandOperationStop);

	// monitoring Battery status

Ton_Delay_BatteryError (In := fbBattery.stDataXelectrix.eErrorState =2,
						PT :=T#5S,
						Q => m_BatteryErrorActive);

Ton_Delay_BatteryModbusError (	In := fbBattery.stDataXelectrix.eErrorState = 1,
								PT :=T#10M,
								Q => m_BatteryModbusCommError);						

Ton_Delay_BatterySPError (	In := ABS(fbBattery.iSetpointPower/10-lrPowerBattery) > 20 AND fbBattery.stDataXelectrix.eGridState<>2 AND fbBattery.stDataBatt.dwSOC<90,	// not alarming during island operation
							PT :=T#1m,
							Q => m_BatteryTargetSPError);	
							
b_Battery_ModbusFault := fbBattery.stDataXelectrix.eErrorState = 1;

END_PROGRAM

// ---- POUs/prgEM.TcPOU
PROGRAM prgEM
VAR
	fbKBusState		: FB_K_Bus_State;
	fbEM1			: FB_EM_Beckhoff_KL3403;
	bHouseEnabled	: BOOL;								//{#lynus.ag#()}
	lrPowerHouse	: LREAL;							//{#lynus.ag#()}
	lrPowerEM1_1	: LREAL;							//{#lynus.ag#()}
	lrPowerEM1_2	: LREAL;							//{#lynus.ag#()}
	lrPowerEM1_3	: LREAL;							//{#lynus.ag#()}
	lrCounterHouse	: LREAL;							//{#lynus.ag#()}
	// Virtual House Test
	fbVirtHouse				: FB_HouseC_Power_Virtual;
	bVirtHouseEnabled		: BOOL;							//{#lynus.ag#()}
	lrPowerVirtHouse		: LREAL;						//{#lynus.ag#()}
	r_PF1	:REAL;
	r_PF2	:REAL;
	r_PF3	:REAL;
	
	r_P_L1: LREAL;
	r_P_L2: LREAL;
	r_P_L3: LREAL;	
	uint_KBusState		:UINT;							//{#lynus.ag#()}
	lrPowerHouseCalculated: LREAL;							//{#lynus.ag#()}
	
	// Sub-Meter for selling energy to local tenant
	fbSubMeter_1				: FB_ENERGYMID_EM22xx_23xx;
	lrPower_SM1				    : LREAL;      //{#lynus.ag#()}
	lrPower_SM1_L1				: LREAL;      //{#lynus.ag#()}
	lrPower_SM1_L2				: LREAL;      //{#lynus.ag#()}
	lrPower_SM1_L3				: LREAL;      //{#lynus.ag#()}
	lrReactivePower_SM1			: LREAL;      //{#lynus.ag#()}
	lrReactivePower_SM1_L1	  	: LREAL;      //{#lynus.ag#()}
	lrReactivePower_SM1_L2	  	: LREAL;      //{#lynus.ag#()}
	lrReactivePower_SM1_L3	  	: LREAL;      //{#lynus.ag#()}
	lrPowerFactor_SM1			: LREAL;      //{#lynus.ag#()}
	lrPowerFactor_SM1_L1		: LREAL;      //{#lynus.ag#()}
	lrPowerFactor_SM1_L2		: LREAL;      //{#lynus.ag#()}
	lrPowerFactor_SM1_L3		: LREAL;      //{#lynus.ag#()}
	lrFrequency_SM1				: LREAL;      //{#lynus.ag#()}
	lrVoltage_SM1_L1N_V		    : LREAL;      //{#lynus.ag#()}
	lrVoltage_SM1_L2N_V		    : LREAL;      //{#lynus.ag#()}
	lrVoltage_SM1_L3N_V		    : LREAL;      //{#lynus.ag#()}
	lrVoltage_SM1_L1L2_V		: LREAL;      //{#lynus.ag#()}
	lrVoltage_SM1_L2L3_V		: LREAL;      //{#lynus.ag#()}
	lrVoltage_SM1_L3L1_V		: LREAL;      //{#lynus.ag#()}
	lrCurrent_SM1_L1			: LREAL;      //{#lynus.ag#()}
	lrCurrent_SM1_L2			: LREAL;      //{#lynus.ag#()}
	lrCurrent_SM1_L3			: LREAL;      //{#lynus.ag#()}
	lrEnergyTotal_Import_SM1	: LREAL;      //{#lynus.ag#()}
	lrEnergyTotal_Export_SM1	: LREAL;      //{#lynus.ag#()}
END_VAR
VAR PERSISTENT
	bEnableHouse		: BOOL;							//{#lynus.ag#()}
	bEnableVirtHouse	: BOOL;							//{#lynus.ag#()}
END_VAR

//The mapping of this function must be linked with the K-Bus State in the E/A Part
fbKBusState(	uiKBusState_OUT=> , 
				b_Kbus_notOk=> , 
				word_ErrorCount=> );

//The mapping of this function must be linked with the KL3403 in the E/A Part
//UV1
fbEM1(
	bEnable:= bEnableHouse, 
	bChannel1Invers:= FALSE,				//Invert power data when transformer are mounted upside down
	bChannel2Invers:= FALSE,			// CT seems to be wired the wrong wy around
	bChannel3Invers:= FALSE,
	uiCurrentTransformerRatioL1:= 400, //Transformer ratio on the secondary side
	uiCurrentTransformerRatioL2:= 400, 
	uiCurrentTransformerRatioL3:= 400, 
	uiKBusState_IN:= fbKBusState.uiKBusState_OUT, 
	stDataEMPower=> , 
	stDataEMCounter=> , 
	stDataEMPowerRealTime=> , 
	stDataEMCounterRealTime=> , 
	diNrOfEM_OUT=> );
	
uint_KBusState :=	fbKBusState.uiKBusState_OUT;

r_PF1 := FBEM1.stDataL1.rPowerfactor;
r_PF2 := FBEM1.stDataL2.rPowerfactor;
r_PF3 := FBEM1.stDataL3.rPowerfactor;
r_P_L1	:= FBEM1.stDataL1.rPower/1000;
r_P_L2	:= FBEM1.stDataL2.rPower/1000;
r_P_L3	:= FBEM1.stDataL3.rPower/1000;

lrPowerHouse := fbEM1.stDataEMPower.lrPowerTotal;
	lrCounterHouse := fbEM1.stDataEMCounter.lrTotalCounterEnergy_Consumption;	
		lrPowerEM1_1 := fbEM1.stDataEMPower.lrPowerL1;
			lrPowerEM1_2 := fbEM1.stDataEMPower.lrPowerL2;
				lrPowerEM1_3 := fbEM1.stDataEMPower.lrPowerL3;
					bHouseEnabled := fbEM1.bEnable;

// VirtualHouse, as Reference to EM Measurement
fbVirtHouse(
	bEnable:= bEnableVirtHouse, 
	diNrOfEMS_IN:= prgEMS.fbEMS.diNrOfEMS_OUT, 
	bSetDefault:= , 
	lrCounterConsumptionSetDefault:= , 
	lrCounterProductionSetDefault:= , 
	stDataHouseC=> , 
	diNrOfHouseC_OUT=> );
	
lrPowerVirtHouse := lrPowerHouseCalculated;		//fbVirtHouse.stDataHouseC.lrPower-prgCS.lrPowerCS;
	bVirtHouseEnabled := fbVirtHouse.stDataHouseC.bEnabled;
	
lrPowerHouseCalculated := MAX(0,prgEM.fbEM1.stDataEMPowerRealTime.lrPowerTotal + prgPV.lrPowerPV + prgBattery.lrPowerBattery - prgCS.lrPowerCS);


// Sub-Meter (for selling energy to local tenant)

fbSubMeter_1(
	m_Enable:= TRUE, 
	str_IPAdress:= '192.168.0.105', 
	real_RealPower_kW => lrPower_SM1,
	real_RealPowerL1_kW => lrPower_SM1_L1,
	real_RealPowerL2_kW => lrPower_SM1_L2,
	real_RealPowerL3_kW => lrPower_SM1_L3,
	real_ReactivePowerL1_kVAr => lrReactivePower_SM1_L1,
	real_ReactivePowerL2_kVAr => lrReactivePower_SM1_L2,
	real_ReactivePowerL3_kVAr => lrReactivePower_SM1_L3,
	real_ReactivePower_kVAr => lrReactivePower_SM1,
	real_PowerFactorL1 => lrPowerFactor_SM1_L1,
	real_PowerFactorL2 => lrPowerFactor_SM1_L2,
	real_PowerFactorL3 => lrPowerFactor_SM1_L3,
	real_PowerFactor => lrPowerFactor_SM1,
	real_Frequency_Hz => lrFrequency_SM1,
	real_VoltageL1N_V => lrVoltage_SM1_L1N_V,
	real_VoltageL2N_V => lrVoltage_SM1_L2N_V,
	real_VoltageL3N_V => lrVoltage_SM1_L3N_V,
	real_VoltageL1L2_V => lrVoltage_SM1_L1L2_V,
	real_VoltageL2L3_V => lrVoltage_SM1_L2L3_V,
	real_VoltageL3L1_V => lrVoltage_SM1_L3L1_V,
	real_CurrentL1_A => lrCurrent_SM1_L1,
	real_CurrentL2_A => lrCurrent_SM1_L2,
	real_CurrentL3_A => lrCurrent_SM1_L3,
	real_EnergyTotal_Import_kWh => lrEnergyTotal_Import_SM1,
	real_EnergyTotal_Export_kWh => lrEnergyTotal_Export_SM1,
	m_PollSuccessful=> , 
	udint_Error_ID=> );

END_PROGRAM

// ---- POUs/prgGrid.TcPOU
PROGRAM prgGrid
VAR PERSISTENT
	rSizeGridConn				: REAL;									//{#lynus.ag#()}
	lrCounterGridProd			: LREAL;								//{#lynus.ag#()}
	lrCounterGridCons			: LREAL;								//{#lynus.ag#()}
END_VAR
VAR
	fbGrid						: FB_Grid_Power;
	fbGridCounter				: FB_EnergyCounter;
	lrGridPower					: LREAL;								//{#lynus.ag#()}
END_VAR

fbGrid(
	bEnable:= TRUE, 
	diNrOfEMS_IN:= prgEMS.fbEMS.diNrOfEMS_OUT, 
	diNrOfEM_IN_Grid:= 	prgEM.fbEM1.diNrOfEM_OUT,			//prgBattery.fbBattery.diNrOfEM_OUT_Grid, 
	rSizeGridConn:= rSizeGridConn, 
	stDataGrid=> , 
	diNrOfGrid_OUT=> );
	
lrGridPower := fbGrid.stDataGrid.lrPower;


// EnergyCounter
fbGridCounter(
	byActiveTariff:= 1, 
	lrPowerInput:= lrGridPower, 
	lrTotalCounterEnergy_Consumption=> , 
	lrTotalCounterEnergy_Production=> , 
	lrCounterEnergyT1_Consumption=> , 
	lrCounterEnergyT2_Consumption=> , 
	lrCounterEnergyT1_Production=> , 
	lrCounterEnergyT2_Production=> );

	IF fbGridCounter.lrTotalCounterEnergy_Production > lrCounterGridProd THEN  	
			lrCounterGridProd := fbGridCounter.lrTotalCounterEnergy_Production;
	END_IF

		IF fbGridCounter.lrTotalCounterEnergy_Consumption > lrCounterGridCons THEN  	
			lrCounterGridCons := fbGridCounter.lrTotalCounterEnergy_Consumption;
		END_IF

END_PROGRAM

// ---- POUs/prgCalc.TcPOU
PROGRAM prgCalc
VAR
	iQuota_Total_PV				: INT;      //{#lynus.ag#()}
	iQuota_Total_Battery		: INT;      //{#lynus.ag#()}
	iQuota_Total_Grid			: INT;      //{#lynus.ag#()}
	iQuota_Total_Sum			: INT;      //{#lynus.ag#()}
	lrPower_TotalConsumption	: LREAL;      //{#lynus.ag#()}

	fbCounter_SM1_PV			: FB_EnergyCounter;
	fbCounter_SM1_Battery		: FB_EnergyCounter;
	fbCounter_SM1_Grid			: FB_EnergyCounter;
	fbCounter_SM1_Total			: FB_EnergyCounter;
	lrPower_SM1_quota_PV		: LREAL;      //{#lynus.ag#()}
	lrPower_SM1_quota_Battery	: LREAL;      //{#lynus.ag#()}
	lrPower_SM1_quota_Grid		: LREAL;      //{#lynus.ag#()}
	
	lrPower_House_quota_PV		: LREAL;      //{#lynus.ag#()}
	lrPower_House_quota_Battery	: LREAL;      //{#lynus.ag#()}
	lrPower_House_quota_Grid		: LREAL;      //{#lynus.ag#()}
END_VAR
VAR PERSISTENT
	lrCounter_SM1_PV		: LREAL;      //{#lynus.ag#()}
	lrCounter_SM1_Battery	: LREAL;      //{#lynus.ag#()}
	lrCounter_SM1_Grid		: LREAL;      //{#lynus.ag#()}
	lrCounter_SM1_Total		: LREAL;      //{#lynus.ag#()}
END_VAR

// calc overall Energymix percentage stakes

lrPower_TotalConsumption := LIMIT(0.001,(LIMIT(0,prgGrid.lrGridPower,9999) + prgPV.lrPowerPV + LIMIT(0,prgBattery.lrPowerBattery,9999)),9999);
iQuota_Total_PV := LREAL_TO_INT((prgPV.lrPowerPV * 100) / lrPower_TotalConsumption);

IF prgBattery.lrPowerBattery > 0 THEN  	
	iQuota_Total_Battery := LREAL_TO_INT((prgBattery.lrPowerBattery * 100) / lrPower_TotalConsumption);
ELSE
	iQuota_Total_Battery := 0;
END_IF

IF prgGrid.lrGridPower > 0 THEN  	
	iQuota_Total_Grid := LREAL_TO_INT((prgGrid.lrGridPower * 100) / lrPower_TotalConsumption);
ELSE
	iQuota_Total_Grid := 0;
END_IF

iQuota_Total_Sum := iQuota_Total_PV + iQuota_Total_Battery + iQuota_Total_Grid;

// calc Energymix for SM1
lrPower_SM1_quota_PV := prgEM.lrPower_SM1 * (iQuota_Total_PV/100);
lrPower_SM1_quota_Battery := prgEM.lrPower_SM1 * (iQuota_Total_Battery/100);
lrPower_SM1_quota_Grid := prgEM.lrPower_SM1 * (iQuota_Total_Grid/100);

fbCounter_SM1_PV(
	byActiveTariff:= 1, 
	lrPowerInput:= lrPower_SM1_quota_PV, 
	lrTotalCounterEnergy_Consumption=> , 
	lrTotalCounterEnergy_Production=> , 
	lrCounterEnergyT1_Consumption=> , 
	lrCounterEnergyT2_Consumption=> , 
	lrCounterEnergyT1_Production=> , 
	lrCounterEnergyT2_Production=> );
	
IF fbCounter_SM1_PV.lrTotalCounterEnergy_Consumption > lrCounter_SM1_PV THEN  	
	lrCounter_SM1_PV := fbCounter_SM1_PV.lrTotalCounterEnergy_Consumption;
END_IF

fbCounter_SM1_Battery(
	byActiveTariff:= 1, 
	lrPowerInput:= lrPower_SM1_quota_Battery, 
	lrTotalCounterEnergy_Consumption=> , 
	lrTotalCounterEnergy_Production=> , 
	lrCounterEnergyT1_Consumption=> , 
	lrCounterEnergyT2_Consumption=> , 
	lrCounterEnergyT1_Production=> , 
	lrCounterEnergyT2_Production=> );
	
IF fbCounter_SM1_Battery.lrTotalCounterEnergy_Consumption > lrCounter_SM1_Battery THEN  	
	lrCounter_SM1_Battery := fbCounter_SM1_Battery.lrTotalCounterEnergy_Consumption;
END_IF

fbCounter_SM1_Grid(
	byActiveTariff:= 1, 
	lrPowerInput:= lrPower_SM1_quota_Grid, 
	lrTotalCounterEnergy_Consumption=> , 
	lrTotalCounterEnergy_Production=> , 
	lrCounterEnergyT1_Consumption=> , 
	lrCounterEnergyT2_Consumption=> , 
	lrCounterEnergyT1_Production=> , 
	lrCounterEnergyT2_Production=> );
	
IF fbCounter_SM1_Grid.lrTotalCounterEnergy_Consumption > lrCounter_SM1_Grid THEN  	
	lrCounter_SM1_Grid := fbCounter_SM1_Grid.lrTotalCounterEnergy_Consumption;
END_IF

// calc Energymix for House
lrPower_House_quota_PV := prgEM.lrPowerVirtHouse * (iQuota_Total_PV/100);
lrPower_House_quota_Battery := prgEM.lrPowerVirtHouse * (iQuota_Total_Battery/100);
lrPower_House_quota_Grid := prgEM.lrPowerVirtHouse * (iQuota_Total_Battery/100);

END_PROGRAM

// ---- POUs/prgComEffIO.TcPOU
PROGRAM prgComEffIO
VAR
	fbCom		: FB_MqttCommunicator_V3;
END_VAR

fbCom(
	bConnect:= TRUE, 
	strAuthKey:=  'BMS99299754422' , 
	sUserName:= '9c801c0d-8c2c-4278-a890-f6835690b001', 
	sUserPassword:= '4eabb1b6-b62b-40a2-976a-790462614f0c', 
	eSavePositionCertificate:= eSavePositionOnPLC.ePostionHardDisk, 
	time_HeartBeat_sec 		:= T#15S,
	bConnected=> , 
	bError=> , 
	hrErrorCode=> , 
	eConnectionState=> , 
	eErrorMessage_Out=> );
(* old
	sUserName:= '42ed263c-2a5f-4093-831d-18453bb20ab2', 
	sUserPassword:= '1dfb7dd2-4ea2-4174-bf5e-9fabdb42463b', 

	*)

END_PROGRAM

// ---- FB/FB_ModBus_100Registers_FC3.TcPOU
FUNCTION_BLOCK FB_ModBus_100Registers_FC3
VAR_INPUT PERSISTENT
	m_Enable					: BOOL;						//Enable the Fuctionblock and his logic
	str_IPAdress				: STRING(15);				//IP Adress of the meter
	w_Adress					: WORD;						//modbus adress
	usint_Quantity				: USINT;					//Number of Words to get polled, max 100
	b_UnitID					: BYTE;						//unitID
END_VAR
VAR_OUTPUT
	m_PollSuccessful			: BOOL;						//Poll succesfull		
	w_Array_Received			: ARRAY[1..100] OF WORD;	// received data
	udint_Error_ID				: UDINT;					// ERR ID FB_MBReadRegs
END_VAR
VAR
	
	timer_Delay					: TON;						//Timer for Delay between Requests
	
	timer_DelayStart			: TON;						//Timer to start the state machine with Delay after enabling or after the system ist restartet
	
	timer_TimeOut				: TON;						//Timer for Timeout MB Read
	
	iStateModbusRead			: INT;						//State machine for read out Data over Modbus RTU
	
	fbMBRead_FC3				: FB_MBReadRegs  ;		//Modbus Read Function (FC3)
	
	ftrig_PEnable				: f_trig;					//Internal positive Edge
	
	iStateModbusError			: INT;						//State machine for error out Data over Modbus TCP/IP	
	
	FPError_FC_3				: R_TRIG;					//Internal positive Edge
	
	arrBuffer_FC3				: ARRAY[1..100] OF WORD;		//Buffer with Data from FC3
	
	timer_Connection_ok			: TON;
	int_Data_Received			: INT;
	
	m_MBTCPError				: BOOL;
	
	int_Data_Received_old		: INT;
	
	timer_Connection_ok_TOF	: TOF;
	
	fbConvertWordToDword		: FB_CV_WORD_TO_DWORD;			//Convert Word to Dword
	
	m_Poll_ok: BOOL;
	
	timer_Wait: Ton;
	int_TimeoutError: INT;
	int_FC3Error: INT;

END_VAR

(*	{attribute 'hide'}--------------------------------------------------------------------------------------------Limits-------------------------------------------------------------------------------------*)

w_Adress := LIMIT(0,w_Adress,60000);
usint_Quantity := LIMIT(1,usint_Quantity,100);
b_UnitID := LIMIT(0,b_UnitID,254);
	
(*--------------------------------------------------------------------------------------------State Machine Read--------------------------------------------------------------------------------------*)

//Timer for Delay
timer_Delay(IN:= , PT:= T#50MS, Q=> , ET=> );

//Timeout Timer is dissabled when the Init Step is aktiv or the function is not enabled
IF iStateModbusRead = 0 OR NOT m_Enable THEN 
	timer_Timeout.IN := FALSE; 
END_IF
timer_Timeout(IN:= , PT:= T#1S, Q=> , ET=> );

